  Call Extruder(272.17524)
  MoveL 6100 to (227.15, 164.34, 88.06) mm, rotated rx 180 ry 0 rz 180 deg; joints [-30.903, 18.099, 54.936, 64.012, 34.845, -59.291]
  MoveL 6101 to (227.15, 164.34, 88.06) mm, rotated rx 180 ry 0 rz 180 deg; joints [-30.903, 18.099, 54.936, 64.012, 34.845, -59.291]
  Call Extruder(272.32310)
  MoveL 6102 to (226.87, 164.39, 88.06) mm, rotated rx 180 ry 0 rz 180 deg; joints [-30.923, 18.056, 54.993, 64.047, 34.856, -59.326]
  MoveL 6103 to (226.87, 164.39, 88.06) mm, rotated rx 180 ry 0 rz 180 deg; joints [-30.923, 18.056, 54.993, 64.047, 34.856, -59.326]
  Call Extruder(272.48484)
  MoveL 6104 to (226.57, 164.44, 88.06) mm, rotated rx 180 ry 0 rz 180 deg; joints [-30.943, 18.008, 55.056, 64.085, 34.867, -59.365]
  MoveL 6105 to (226.57, 164.44, 88.06) mm, rotated rx 180 ry 0 rz 180 deg; joints [-30.943, 18.008, 55.056, 64.085, 34.867, -59.365]
  Call Extruder(272.64586)
  MoveL 6106 to (226.26, 164.49, 88.06) mm, rotated rx 180 ry 0 rz 180 deg; joints [-30.964, 17.96, 55.119, 64.122, 34.879, -59.404]
  MoveL 6107 to (226.26, 164.49, 88.06) mm, rotated rx 180 ry 0 rz 180 deg; joints [-30.964, 17.96, 55.119, 64.122, 34.879, -59.404]
  Call Extruder(272.80614)
  MoveL 6108 to (225.95, 164.53, 88.06) mm, rotated rx 180 ry 0 rz 180 deg; joints [-30.985, 17.912, 55.182, 64.16, 34.89, -59.442]
  MoveL 6109 to (225.95, 164.53, 88.06) mm, rotated rx 180 ry 0 rz 180 deg; joints [-30.985, 17.912, 55.182, 64.16, 34.89, -59.442]
  Call Extruder(272.96570)
  MoveL 6110 to (225.65, 164.58, 88.06) mm, rotated rx 180 ry 0 rz 180 deg; joints [-31.006, 17.864, 55.244, 64.198, 34.901, -59.481]
  MoveL 6111 to (225.65, 164.58, 88.06) mm, rotated rx 180 ry 0 rz 180 deg; joints [-31.006, 17.864, 55.244, 64.198, 34.901, -59.481]
  Call Extruder(273.12452)
  MoveL 6112 to (225.34, 164.63, 88.06) mm, rotated rx -180 ry 0 rz 180 deg; joints [-31.027, 17.817, 55.307, 64.235, 34.913, -59.519]
  MoveL 6113 to (225.34, 164.63, 88.06) mm, rotated rx -180 ry 0 rz 180 deg; joints [-31.027, 17.817, 55.307, 64.235, 34.913, -59.519]
  Call Extruder(273.30319)
  MoveL 6114 to (225, 164.68, 88.06) mm, rotated rx 180 ry 0 rz 180 deg; joints [-31.049, 17.762, 55.379, 64.278, 34.925, -59.563]
  MoveL 6115 to (225, 164.68, 88.06) mm, rotated rx 180 ry 0 rz 180 deg; joints [-31.049, 17.762, 55.379, 64.278, 34.925, -59.563]
  Call Extruder(273.50164)
  MoveL 6116 to (224.61, 164.72, 88.06) mm, rotated rx -180 ry 0 rz 180 deg; joints [-31.074, 17.7, 55.459, 64.324, 34.939, -59.611]
  MoveL 6117 to (224.61, 164.72, 88.06) mm, rotated rx -180 ry 0 rz 180 deg; joints [-31.074, 17.7, 55.459, 64.324, 34.939, -59.611]
  Call Extruder(273.69921)
  MoveL 6118 to (224.22, 164.77, 88.06) mm, rotated rx 180 ry 0 rz 180 deg; joints [-31.1, 17.638, 55.54, 64.371, 34.952, -59.659]
  MoveL 6119 to (224.22, 164.77, 88.06) mm, rotated rx 180 ry 0 rz 180 deg; joints [-31.1, 17.638, 55.54, 64.371, 34.952, -59.659]
  Call Extruder(273.89592)
  MoveL 6120 to (223.84, 164.82, 88.06) mm, rotated rx 180 ry 0 rz 180 deg; joints [-31.125, 17.576, 55.621, 64.417, 34.966, -59.706]
  MoveL 6121 to (223.84, 164.82, 88.06) mm, rotated rx 180 ry 0 rz 180 deg; joints [-31.125, 17.576, 55.621, 64.417, 34.966, -59.706]
  Call Extruder(274.09176)
  MoveL 6122 to (223.45, 164.86, 88.06) mm, rotated rx -180 ry 0 rz 180 deg; joints [-31.15, 17.514, 55.701, 64.463, 34.979, -59.754]
  MoveL 6123 to (223.45, 164.86, 88.06) mm, rotated rx -180 ry 0 rz 180 deg; joints [-31.15, 17.514, 55.701, 64.463, 34.979, -59.754]
  Call Extruder(274.38712)
  MoveL 6124 to (222.86, 164.91, 88.06) mm, rotated rx 180 ry 0 rz -180 deg; joints [-31.186, 17.419, 55.826, 64.533, 34.998, -59.826]
  MoveL 6125 to (222.86, 164.91, 88.06) mm, rotated rx 180 ry 0 rz -180 deg; joints [-31.186, 17.419, 55.826, 64.533, 34.998, -59.826]
  Call Extruder(274.68114)
  MoveL 6126 to (222.27, 164.96, 88.06) mm, rotated rx 180 ry 0 rz 180 deg; joints [-31.222, 17.323, 55.951, 64.601, 35.017, -59.897]
  MoveL 6127 to (222.27, 164.96, 88.06) mm, rotated rx 180 ry 0 rz 180 deg; joints [-31.222, 17.323, 55.951, 64.601, 35.017, -59.897]
  Call Extruder(274.97384)
  MoveL 6128 to (221.68, 165, 88.06) mm, rotated rx 180 ry 0 rz 180 deg; joints [-31.258, 17.227, 56.075, 64.67, 35.036, -59.968]
  MoveL 6129 to (221.68, 165, 88.06) mm, rotated rx 180 ry 0 rz 180 deg; joints [-31.258, 17.227, 56.075, 64.67, 35.036, -59.968]
  Call Extruder(275.54729)
  MoveL 6130 to (220.52, 165.05, 88.06) mm, rotated rx 180 ry 0 rz 180 deg; joints [-31.326, 17.035, 56.324, 64.802, 35.07, -60.106]
  MoveL 6131 to (220.52, 165.05, 88.06) mm, rotated rx 180 ry 0 rz 180 deg; joints [-31.326, 17.035, 56.324, 64.802, 35.07, -60.106]
  Call Extruder(276.26129)
  MoveL 6132 to (219.06, 165.09, 88.06) mm, rotated rx -180 ry 0 rz 180 deg; joints [-31.409, 16.794, 56.636, 64.966, 35.113, -60.277]
  Call Extruder(393.10803)
  MoveL 6133 to (-19.06, 165.09, 88.06) mm, rotated rx 180 ry 0 rz 180 deg; joints [-51.475, -12.583, 87.083, 77.988, 53.116, -70.481]
  Call Extruder(393.53664)
  MoveL 6134 to (-19.94, 165.07, 88.06) mm, rotated rx 180 ry 0 rz 180 deg; joints [-51.582, -12.664, 87.145, 78.02, 53.22, -70.486]
  MoveL 6135 to (-19.94, 165.07, 88.06) mm, rotated rx 180 ry 0 rz 180 deg; joints [-51.582, -12.664, 87.145, 78.02, 53.22, -70.486]
  Call Extruder(394.11009)
  MoveL 6136 to (-21.1, 165.03, 88.06) mm, rotated rx 180 ry 0 rz 180 deg; joints [-51.722, -12.772, 87.23, 78.061, 53.357, -70.492]
  MoveL 6137 to (-21.1, 165.03, 88.06) mm, rotated rx 180 ry 0 rz 180 deg; joints [-51.722, -12.772, 87.23, 78.061, 53.357, -70.492]
  Call Extruder(394.54439)
  MoveL 6138 to (-21.97, 164.98, 88.06) mm, rotated rx 180 ry 0 rz 180 deg; joints [-51.827, -12.855, 87.295, 78.091, 53.46, -70.495]
  MoveL 6139 to (-21.97, 164.98, 88.06) mm, rotated rx 180 ry 0 rz 180 deg; joints [-51.827, -12.855, 87.295, 78.091, 53.46, -70.495]
  Call Extruder(394.83842)
  MoveL 6140 to (-22.56, 164.93, 88.06) mm, rotated rx 180 ry 0 rz -180 deg; joints [-51.897, -12.913, 87.34, 78.111, 53.528, -70.497]
  MoveL 6141 to (-22.56, 164.93, 88.06) mm, rotated rx 180 ry 0 rz -180 deg; joints [-51.897, -12.913, 87.34, 78.111, 53.528, -70.497]
  Call Extruder(395.13378)
  MoveL 6142 to (-23.15, 164.89, 88.06) mm, rotated rx 180 ry 0 rz 180 deg; joints [-51.966, -12.97, 87.384, 78.131, 53.596, -70.499]
  MoveL 6143 to (-23.15, 164.89, 88.06) mm, rotated rx 180 ry 0 rz 180 deg; joints [-51.966, -12.97, 87.384, 78.131, 53.596, -70.499]
  Call Extruder(395.37999)
  MoveL 6144 to (-23.64, 164.84, 88.06) mm, rotated rx 180 ry 0 rz 180 deg; joints [-52.023, -13.018, 87.421, 78.146, 53.652, -70.499]
  MoveL 6145 to (-23.64, 164.84, 88.06) mm, rotated rx 180 ry 0 rz 180 deg; joints [-52.023, -13.018, 87.421, 78.146, 53.652, -70.499]
  Call Extruder(395.57670)
  MoveL 6146 to (-24.03, 164.79, 88.06) mm, rotated rx -180 ry 0 rz 180 deg; joints [-52.067, -13.058, 87.452, 78.158, 53.696, -70.499]
  MoveL 6147 to (-24.03, 164.79, 88.06) mm, rotated rx -180 ry 0 rz 180 deg; joints [-52.067, -13.058, 87.452, 78.158, 53.696, -70.499]
  Call Extruder(395.77427)
  MoveL 6148 to (-24.42, 164.75, 88.06) mm, rotated rx 180 ry 0 rz 180 deg; joints [-52.112, -13.097, 87.482, 78.17, 53.739, -70.5]
  MoveL 6149 to (-24.42, 164.75, 88.06) mm, rotated rx 180 ry 0 rz 180 deg; joints [-52.112, -13.097, 87.482, 78.17, 53.739, -70.5]
  Call Extruder(395.97271)
  MoveL 6150 to (-24.8, 164.7, 88.06) mm, rotated rx 180 ry 0 rz 180 deg; joints [-52.156, -13.136, 87.513, 78.182, 53.783, -70.5]
  MoveL 6151 to (-24.8, 164.7, 88.06) mm, rotated rx 180 ry 0 rz 180 deg; joints [-52.156, -13.136, 87.513, 78.182, 53.783, -70.5]
  Call Extruder(396.17202)
  MoveL 6152 to (-25.19, 164.66, 88.06) mm, rotated rx 180 ry 0 rz 180 deg; joints [-52.2, -13.176, 87.543, 78.194, 53.827, -70.5]
  MoveL 6153 to (-25.19, 164.66, 88.06) mm, rotated rx 180 ry 0 rz 180 deg; joints [-52.2, -13.176, 87.543, 78.194, 53.827, -70.5]
  Call Extruder(396.33085)
  MoveL 6154 to (-25.5, 164.61, 88.06) mm, rotated rx 180 ry 0 rz 180 deg; joints [-52.235, -13.208, 87.568, 78.203, 53.86, -70.499]
  MoveL 6155 to (-25.5, 164.61, 88.06) mm, rotated rx 180 ry 0 rz 180 deg; joints [-52.235, -13.208, 87.568, 78.203, 53.86, -70.499]
  Call Extruder(396.49041)
  MoveL 6156 to (-25.8, 164.56, 88.06) mm, rotated rx 180 ry 0 rz 180 deg; joints [-52.269, -13.24, 87.593, 78.212, 53.894, -70.498]
  MoveL 6157 to (-25.8, 164.56, 88.06) mm, rotated rx 180 ry 0 rz 180 deg; joints [-52.269, -13.24, 87.593, 78.212, 53.894, -70.498]
  Call Extruder(396.65070)
  MoveL 6158 to (-26.11, 164.51, 88.06) mm, rotated rx 180 ry 0 rz -180 deg; joints [-52.303, -13.272, 87.618, 78.221, 53.927, -70.498]
  MoveL 6159 to (-26.11, 164.51, 88.06) mm, rotated rx 180 ry 0 rz -180 deg; joints [-52.303, -13.272, 87.618, 78.221, 53.927, -70.498]
  Call Extruder(396.81172)
  MoveL 6160 to (-26.41, 164.46, 88.06) mm, rotated rx 180 ry 0 rz -180 deg; joints [-52.337, -13.305, 87.643, 78.229, 53.961, -70.497]
  MoveL 6161 to (-26.41, 164.46, 88.06) mm, rotated rx 180 ry 0 rz -180 deg; joints [-52.337, -13.305, 87.643, 78.229, 53.961, -70.497]
  Call Extruder(396.97346)
  MoveL 6162 to (-26.72, 164.41, 88.06) mm, rotated rx -180 ry 0 rz 180 deg; joints [-52.371, -13.337, 87.668, 78.238, 53.995, -70.496]
  MoveL 6163 to (-26.72, 164.41, 88.06) mm, rotated rx -180 ry 0 rz 180 deg; joints [-52.371, -13.337, 87.668, 78.238, 53.995, -70.496]
  Call Extruder(397.13593)
  MoveL 6164 to (-27.02, 164.37, 88.06) mm, rotated rx 180 ry 0 rz -180 deg; joints [-52.405, -13.369, 87.692, 78.247, 54.028, -70.496]
  MoveL 6165 to (-27.02, 164.37, 88.06) mm, rotated rx 180 ry 0 rz -180 deg; joints [-52.405, -13.369, 87.692, 78.247, 54.028, -70.496]
  Call Extruder(397.26986)
  MoveL 6166 to (-27.27, 164.32, 88.06) mm, rotated rx 180 ry 0 rz 180 deg; joints [-52.432, -13.397, 87.713, 78.254, 54.055, -70.495]
  MoveL 6167 to (-27.27, 164.32, 88.06) mm, rotated rx 180 ry 0 rz 180 deg; joints [-52.432, -13.397, 87.713, 78.254, 54.055, -70.495]
  Call Extruder(397.40439)
  MoveL 6168 to (-27.52, 164.27, 88.06) mm, rotated rx 180 ry 0 rz 180 deg; joints [-52.459, -13.424, 87.734, 78.26, 54.082, -70.493]
  MoveL 6169 to (-27.52, 164.27, 88.06) mm, rotated rx 180 ry 0 rz 180 deg; joints [-52.459, -13.424, 87.734, 78.26, 54.082, -70.493]
  Call Extruder(397.53954)
  MoveL 6170 to (-27.77, 164.22, 88.06) mm, rotated rx 180 ry 0 rz 180 deg; joints [-52.486, -13.451, 87.755, 78.267, 54.109, -70.492]
  MoveL 6171 to (-27.77, 164.22, 88.06) mm, rotated rx 180 ry 0 rz 180 deg; joints [-52.486, -13.451, 87.755, 78.267, 54.109, -70.492]
  Call Extruder(397.67530)
  MoveL 6172 to (-28.02, 164.17, 88.06) mm, rotated rx 180 ry 0 rz -180 deg; joints [-52.513, -13.479, 87.776, 78.274, 54.135, -70.491]
  MoveL 6173 to (-28.02, 164.17, 88.06) mm, rotated rx 180 ry 0 rz -180 deg; joints [-52.513, -13.479, 87.776, 78.274, 54.135, -70.491]
  Call Extruder(397.81166)
  MoveL 6174 to (-28.27, 164.12, 88.06) mm, rotated rx 180 ry 0 rz 180 deg; joints [-52.54, -13.506, 87.797, 78.28, 54.162, -70.49]
  MoveL 6175 to (-28.27, 164.12, 88.06) mm, rotated rx 180 ry 0 rz 180 deg; joints [-52.54, -13.506, 87.797, 78.28, 54.162, -70.49]
  Call Extruder(397.89653)
  MoveL 6176 to (-28.43, 164.09, 88.06) mm, rotated rx -180 ry 0 rz -180 deg; joints [-52.556, -13.523, 87.81, 78.284, 54.179, -70.489]
  Set speed (130.0 mm/s)
  MoveL 6177 to (-31.76, 163.31, 88.06) mm, rotated rx 180 ry 0 rz 180 deg; joints [-52.91, -13.899, 88.098, 78.367, 54.529, -70.466]
  MoveL 6178 to (-31.76, 163.31, 97.46) mm, rotated rx 180 ry 0 rz 180 deg; joints [-52.91, -14.605, 90.097, 79.276, 54.279, -72.028]
  Call Extruder(395.89653)
  Set speed (40.0 mm/s)
  MoveL 6179 to (-31.76, 163.31, 97.46) mm, rotated rx 180 ry 0 rz 180 deg; joints [-52.91, -14.605, 90.097, 79.276, 54.279, -72.028]
  Call Extruder(0.00000)
  Set speed (130.0 mm/s)
  MoveL 6180 to (-31.64, 163.21, 97.46) mm, rotated rx 180 ry 0 rz 180 deg; joints [-52.884, -14.606, 90.098, 79.266, 54.254, -72.022]
  Call Extruder(2.00000)
  Set speed (40.0 mm/s)
  MoveL 6181 to (-31.64, 163.21, 97.46) mm, rotated rx 180 ry 0 rz 180 deg; joints [-52.884, -14.606, 90.098, 79.266, 54.254, -72.022]
  Set speed (30.0 mm/s)
  MoveL 6182 to (-31.64, 163.21, 97.46) mm, rotated rx 180 ry 0 rz 180 deg; joints [-52.884, -14.606, 90.098, 79.266, 54.254, -72.022]
  Call Extruder(2.18198)
  MoveL 6183 to (-31.93, 163.09, 97.46) mm, rotated rx -180 ry 0 rz 180 deg; joints [-52.91, -14.645, 90.127, 79.269, 54.281, -72.016]
  MoveL 6184 to (-31.93, 163.09, 97.46) mm, rotated rx -180 ry 0 rz 180 deg; joints [-52.91, -14.645, 90.127, 79.269, 54.281, -72.016]
  Call Extruder(2.36471)
  MoveL 6185 to (-32.22, 162.97, 97.46) mm, rotated rx 180 ry 0 rz 180 deg; joints [-52.936, -14.684, 90.157, 79.272, 54.307, -72.01]
  MoveL 6186 to (-32.22, 162.97, 97.46) mm, rotated rx 180 ry 0 rz 180 deg; joints [-52.936, -14.684, 90.157, 79.272, 54.307, -72.01]
  Call Extruder(2.53513)
  MoveL 6187 to (-32.49, 162.85, 97.46) mm, rotated rx 180 ry 0 rz 180 deg; joints [-52.96, -14.72, 90.184, 79.275, 54.332, -72.004]
  MoveL 6188 to (-32.49, 162.85, 97.46) mm, rotated rx 180 ry 0 rz 180 deg; joints [-52.96, -14.72, 90.184, 79.275, 54.332, -72.004]
  Call Extruder(2.69310)
  MoveL 6189 to (-32.74, 162.74, 97.46) mm, rotated rx 180 ry 0 rz 180 deg; joints [-52.982, -14.754, 90.209, 79.277, 54.354, -71.999]
  MoveL 6190 to (-32.74, 162.74, 97.46) mm, rotated rx 180 ry 0 rz 180 deg; joints [-52.982, -14.754, 90.209, 79.277, 54.354, -71.999]
  Call Extruder(2.85168)
  MoveL 6191 to (-32.99, 162.64, 97.46) mm, rotated rx 180 ry 0 rz 180 deg; joints [-53.004, -14.788, 90.234, 79.279, 54.377, -71.993]
  MoveL 6192 to (-32.99, 162.64, 97.46) mm, rotated rx 180 ry 0 rz 180 deg; joints [-53.004, -14.788, 90.234, 79.279, 54.377, -71.993]
  Call Extruder(3.05785)
  MoveL 6193 to (-33.29, 162.46, 97.46) mm, rotated rx 180 ry 0 rz 180 deg; joints [-53.026, -14.834, 90.269, 79.28, 54.4, -71.984]
  MoveL 6194 to (-33.29, 162.46, 97.46) mm, rotated rx 180 ry 0 rz 180 deg; joints [-53.026, -14.834, 90.269, 79.28, 54.4, -71.984]
  Call Extruder(3.26479)
  MoveL 6195 to (-33.6, 162.29, 97.46) mm, rotated rx 180 ry 0 rz 180 deg; joints [-53.049, -14.88, 90.303, 79.28, 54.424, -71.975]
  MoveL 6196 to (-33.6, 162.29, 97.46) mm, rotated rx 180 ry 0 rz 180 deg; joints [-53.049, -14.88, 90.303, 79.28, 54.424, -71.975]
  Call Extruder(3.47251)
  MoveL 6197 to (-33.9, 162.11, 97.46) mm, rotated rx 180 ry 0 rz 180 deg; joints [-53.071, -14.926, 90.338, 79.28, 54.447, -71.966]
  MoveL 6198 to (-33.9, 162.11, 97.46) mm, rotated rx 180 ry 0 rz 180 deg; joints [-53.071, -14.926, 90.338, 79.28, 54.447, -71.966]
  Call Extruder(3.68101)
  MoveL 6199 to (-34.21, 161.93, 97.46) mm, rotated rx -180 ry 0 rz -180 deg; joints [-53.094, -14.972, 90.372, 79.281, 54.471, -71.957]
  MoveL 6200 to (-34.21, 161.93, 97.46) mm, rotated rx -180 ry 0 rz -180 deg; joints [-53.094, -14.972, 90.372, 79.281, 54.471, -71.957]
  Call Extruder(3.86055)
  MoveL 6201 to (-34.45, 161.76, 97.46) mm, rotated rx 180 ry 0 rz -180 deg; joints [-53.109, -15.013, 90.403, 79.279, 54.487, -71.947]
  MoveL 6202 to (-34.45, 161.76, 97.46) mm, rotated rx 180 ry 0 rz -180 deg; joints [-53.109, -15.013, 90.403, 79.279, 54.487, -71.947]
  Call Extruder(4.19399)
  MoveL 6203 to (-34.9, 161.43, 97.46) mm, rotated rx 180 ry 0 rz 180 deg; joints [-53.135, -15.09, 90.459, 79.275, 54.516, -71.93]
  MoveL 6204 to (-34.9, 161.43, 97.46) mm, rotated rx 180 ry 0 rz 180 deg; joints [-53.135, -15.09, 90.459, 79.275, 54.516, -71.93]
  Call Extruder(4.52861)
  MoveL 6205 to (-35.35, 161.1, 97.46) mm, rotated rx 180 ry 0 rz 180 deg; joints [-53.163, -15.166, 90.516, 79.272, 54.546, -71.912]
  Call Extruder(5.35652)
  MoveL 6206 to (-36.39, 160.19, 97.46) mm, rotated rx 180 ry 0 rz 180 deg; joints [-53.209, -15.359, 90.659, 79.255, 54.599, -71.862]
  Call Extruder(6.18445)
  MoveL 6207 to (-37.3, 159.15, 97.46) mm, rotated rx 180 ry 0 rz 180 deg; joints [-53.227, -15.555, 90.803, 79.225, 54.626, -71.803]
  Call Extruder(6.35176)
  MoveL 6208 to (-37.47, 158.93, 97.46) mm, rotated rx 180 ry 0 rz 180 deg; joints [-53.227, -15.595, 90.832, 79.218, 54.628, -71.79]
  MoveL 6209 to (-37.47, 158.93, 97.46) mm, rotated rx 180 ry 0 rz 180 deg; joints [-53.227, -15.595, 90.832, 79.218, 54.628, -71.79]
  Call Extruder(6.68519)
  MoveL 6210 to (-37.79, 158.48, 97.46) mm, rotated rx -180 ry 0 rz 180 deg; joints [-53.226, -15.674, 90.89, 79.203, 54.63, -71.765]
  MoveL 6211 to (-37.79, 158.48, 97.46) mm, rotated rx -180 ry 0 rz 180 deg; joints [-53.226, -15.674, 90.89, 79.203, 54.63, -71.765]
  Call Extruder(7.01743)
  MoveL 6212 to (-38.12, 158.03, 97.46) mm, rotated rx 180 ry 0 rz 180 deg; joints [-53.224, -15.754, 90.949, 79.187, 54.633, -71.739]
  MoveL 6213 to (-38.12, 158.03, 97.46) mm, rotated rx 180 ry 0 rz 180 deg; joints [-53.224, -15.754, 90.949, 79.187, 54.633, -71.739]
  Call Extruder(7.13511)
  MoveL 6214 to (-38.22, 157.85, 97.46) mm, rotated rx 180 ry 0 rz 180 deg; joints [-53.221, -15.782, 90.969, 79.181, 54.631, -71.729]
  MoveL 6215 to (-38.22, 157.85, 97.46) mm, rotated rx 180 ry 0 rz 180 deg; joints [-53.221, -15.782, 90.969, 79.181, 54.631, -71.729]
  Call Extruder(7.34283)
  MoveL 6216 to (-38.4, 157.55, 97.46) mm, rotated rx -180 ry 0 rz 180 deg; joints [-53.214, -15.831, 91.005, 79.169, 54.627, -71.711]
  MoveL 6217 to (-38.4, 157.55, 97.46) mm, rotated rx -180 ry 0 rz 180 deg; joints [-53.214, -15.831, 91.005, 79.169, 54.627, -71.711]
  Call Extruder(7.54978)
  MoveL 6218 to (-38.57, 157.25, 97.46) mm, rotated rx 180 ry 0 rz 180 deg; joints [-53.207, -15.881, 91.042, 79.157, 54.623, -71.693]
  MoveL 6219 to (-38.57, 157.25, 97.46) mm, rotated rx 180 ry 0 rz 180 deg; joints [-53.207, -15.881, 91.042, 79.157, 54.623, -71.693]
  Call Extruder(7.75595)
  MoveL 6220 to (-38.75, 156.94, 97.46) mm, rotated rx 180 ry 0 rz 180 deg; joints [-53.2, -15.93, 91.078, 79.144, 54.619, -71.676]
  MoveL 6221 to (-38.75, 156.94, 97.46) mm, rotated rx 180 ry 0 rz 180 deg; joints [-53.2, -15.93, 91.078, 79.144, 54.619, -71.676]
  Call Extruder(7.93762)
  MoveL 6222 to (-38.89, 156.67, 97.46) mm, rotated rx 180 ry 0 rz 180 deg; joints [-53.191, -15.974, 91.109, 79.133, 54.613, -71.659]
  MoveL 6223 to (-38.89, 156.67, 97.46) mm, rotated rx 180 ry 0 rz 180 deg; joints [-53.191, -15.974, 91.109, 79.133, 54.613, -71.659]
  Call Extruder(8.09561)
  MoveL 6224 to (-39, 156.42, 97.46) mm, rotated rx 180 ry 0 rz 180 deg; joints [-53.18, -16.011, 91.137, 79.122, 54.605, -71.645]
  MoveL 6225 to (-39, 156.42, 97.46) mm, rotated rx 180 ry 0 rz 180 deg; joints [-53.18, -16.011, 91.137, 79.122, 54.605, -71.645]
  Call Extruder(8.25299)
  MoveL 6226 to (-39.1, 156.17, 97.46) mm, rotated rx 180 ry 0 rz 180 deg; joints [-53.17, -16.049, 91.164, 79.11, 54.596, -71.63]
  MoveL 6227 to (-39.1, 156.17, 97.46) mm, rotated rx 180 ry 0 rz 180 deg; joints [-53.17, -16.049, 91.164, 79.11, 54.596, -71.63]
  Call Extruder(8.43571)
  MoveL 6228 to (-39.23, 155.88, 97.46) mm, rotated rx 180 ry 0 rz 180 deg; joints [-53.156, -16.092, 91.195, 79.097, 54.586, -71.613]
  MoveL 6229 to (-39.23, 155.88, 97.46) mm, rotated rx 180 ry 0 rz 180 deg; joints [-53.156, -16.092, 91.195, 79.097, 54.586, -71.613]
  Call Extruder(8.61768)
  MoveL 6230 to (-39.35, 155.58, 97.46) mm, rotated rx 180 ry 0 rz 180 deg; joints [-53.143, -16.136, 91.227, 79.083, 54.576, -71.595]
  MoveL 6231 to (-39.35, 155.58, 97.46) mm, rotated rx 180 ry 0 rz 180 deg; joints [-53.143, -16.136, 91.227, 79.083, 54.576, -71.595]
  Call Extruder(8.76501)
  MoveL 6232 to (-39.44, 155.34, 97.46) mm, rotated rx 180 ry 0 rz 180 deg; joints [-53.131, -16.171, 91.252, 79.072, 54.566, -71.581]
  MoveL 6233 to (-39.44, 155.34, 97.46) mm, rotated rx 180 ry 0 rz 180 deg; joints [-53.131, -16.171, 91.252, 79.072, 54.566, -71.581]
  Call Extruder(8.87824)
  MoveL 6234 to (-39.5, 155.15, 97.46) mm, rotated rx 180 ry 0 rz 180 deg; joints [-53.121, -16.198, 91.272, 79.063, 54.558, -71.57]
  MoveL 6235 to (-39.5, 155.15, 97.46) mm, rotated rx 180 ry 0 rz 180 deg; joints [-53.121, -16.198, 91.272, 79.063, 54.558, -71.57]
  Call Extruder(8.99103)
  MoveL 6236 to (-39.56, 154.97, 97.46) mm, rotated rx 180 ry 0 rz 180 deg; joints [-53.11, -16.224, 91.291, 79.053, 54.549, -71.558]
  MoveL 6237 to (-39.56, 154.97, 97.46) mm, rotated rx 180 ry 0 rz 180 deg; joints [-53.11, -16.224, 91.291, 79.053, 54.549, -71.558]
  Call Extruder(9.10338)
  MoveL 6238 to (-39.62, 154.78, 97.46) mm, rotated rx -180 ry 0 rz -180 deg; joints [-53.099, -16.251, 91.31, 79.044, 54.54, -71.547]
  MoveL 6239 to (-39.62, 154.78, 97.46) mm, rotated rx -180 ry 0 rz -180 deg; joints [-53.099, -16.251, 91.31, 79.044, 54.54, -71.547]
  Call Extruder(9.21528)
  MoveL 6240 to (-39.68, 154.59, 97.46) mm, rotated rx 180 ry 0 rz 180 deg; joints [-53.088, -16.277, 91.329, 79.035, 54.531, -71.536]
  MoveL 6241 to (-39.68, 154.59, 97.46) mm, rotated rx 180 ry 0 rz 180 deg; joints [-53.088, -16.277, 91.329, 79.035, 54.531, -71.536]
  Call Extruder(9.33668)
  MoveL 6242 to (-39.75, 154.38, 97.46) mm, rotated rx -180 ry 0 rz 180 deg; joints [-53.076, -16.306, 91.35, 79.024, 54.521, -71.523]
  MoveL 6243 to (-39.75, 154.38, 97.46) mm, rotated rx -180 ry 0 rz 180 deg; joints [-53.076, -16.306, 91.35, 79.024, 54.521, -71.523]
  Call Extruder(9.46747)
  MoveL 6244 to (-39.81, 154.16, 97.46) mm, rotated rx 180 ry 0 rz 180 deg; joints [-53.063, -16.337, 91.373, 79.013, 54.51, -71.51]
  MoveL 6245 to (-39.81, 154.16, 97.46) mm, rotated rx 180 ry 0 rz 180 deg; joints [-53.063, -16.337, 91.373, 79.013, 54.51, -71.51]
  Call Extruder(9.59770)
  MoveL 6246 to (-39.88, 153.94, 97.46) mm, rotated rx 180 ry 0 rz 180 deg; joints [-53.049, -16.368, 91.395, 79.002, 54.499, -71.496]
  MoveL 6247 to (-39.88, 153.94, 97.46) mm, rotated rx 180 ry 0 rz 180 deg; joints [-53.049, -16.368, 91.395, 79.002, 54.499, -71.496]
  Call Extruder(9.72737)
  MoveL 6248 to (-39.95, 153.71, 97.46) mm, rotated rx -180 ry 0 rz -180 deg; joints [-53.036, -16.4, 91.417, 78.99, 54.488, -71.482]
  MoveL 6249 to (-39.95, 153.71, 97.46) mm, rotated rx -180 ry 0 rz -180 deg; joints [-53.036, -16.4, 91.417, 78.99, 54.488, -71.482]
  Call Extruder(9.85647)
  MoveL 6250 to (-40.02, 153.49, 97.46) mm, rotated rx -180 ry 0 rz 180 deg; joints [-53.022, -16.431, 91.44, 78.979, 54.476, -71.469]
  MoveL 6251 to (-40.02, 153.49, 97.46) mm, rotated rx -180 ry 0 rz 180 deg; joints [-53.022, -16.431, 91.44, 78.979, 54.476, -71.469]
  Call Extruder(9.97155)
  MoveL 6252 to (-40.06, 153.28, 97.46) mm, rotated rx 180 ry 0 rz 180 deg; joints [-53.007, -16.458, 91.459, 78.968, 54.464, -71.456]
  MoveL 6253 to (-40.06, 153.28, 97.46) mm, rotated rx 180 ry 0 rz 180 deg; joints [-53.007, -16.458, 91.459, 78.968, 54.464, -71.456]
  Call Extruder(10.08619)
  MoveL 6254 to (-40.11, 153.08, 97.46) mm, rotated rx 180 ry 0 rz 180 deg; joints [-52.993, -16.485, 91.479, 78.957, 54.452, -71.444]
  MoveL 6255 to (-40.11, 153.08, 97.46) mm, rotated rx 180 ry 0 rz 180 deg; joints [-52.993, -16.485, 91.479, 78.957, 54.452, -71.444]
  Call Extruder(10.20037)
  MoveL 6256 to (-40.15, 152.88, 97.46) mm, rotated rx 180 ry 0 rz 180 deg; joints [-52.978, -16.512, 91.498, 78.946, 54.439, -71.431]
  MoveL 6257 to (-40.15, 152.88, 97.46) mm, rotated rx 180 ry 0 rz 180 deg; joints [-52.978, -16.512, 91.498, 78.946, 54.439, -71.431]
  Call Extruder(10.31410)
  MoveL 6258 to (-40.2, 152.67, 97.46) mm, rotated rx -180 ry 0 rz 180 deg; joints [-52.963, -16.539, 91.517, 78.935, 54.426, -71.419]
  MoveL 6259 to (-40.2, 152.67, 97.46) mm, rotated rx -180 ry 0 rz 180 deg; joints [-52.963, -16.539, 91.517, 78.935, 54.426, -71.419]
  Call Extruder(10.43952)
  MoveL 6260 to (-40.24, 152.45, 97.46) mm, rotated rx -180 ry 0 rz 180 deg; joints [-52.946, -16.568, 91.539, 78.922, 54.412, -71.405]
  MoveL 6261 to (-40.24, 152.45, 97.46) mm, rotated rx -180 ry 0 rz 180 deg; joints [-52.946, -16.568, 91.539, 78.922, 54.412, -71.405]
  Call Extruder(10.57650)
  MoveL 6262 to (-40.29, 152.2, 97.46) mm, rotated rx -180 ry 0 rz 180 deg; joints [-52.928, -16.601, 91.562, 78.908, 54.396, -71.39]
  MoveL 6263 to (-40.29, 152.2, 97.46) mm, rotated rx -180 ry 0 rz 180 deg; joints [-52.928, -16.601, 91.562, 78.908, 54.396, -71.39]
  Call Extruder(10.71287)
  MoveL 6264 to (-40.34, 151.95, 97.46) mm, rotated rx -180 ry 0 rz -180 deg; joints [-52.909, -16.633, 91.585, 78.894, 54.38, -71.374]
  MoveL 6265 to (-40.34, 151.95, 97.46) mm, rotated rx -180 ry 0 rz -180 deg; joints [-52.909, -16.633, 91.585, 78.894, 54.38, -71.374]
  Call Extruder(10.84862)
  MoveL 6266 to (-40.39, 151.7, 97.46) mm, rotated rx 180 ry 0 rz 180 deg; joints [-52.89, -16.665, 91.608, 78.881, 54.364, -71.359]
  MoveL 6267 to (-40.39, 151.7, 97.46) mm, rotated rx 180 ry 0 rz 180 deg; joints [-52.89, -16.665, 91.608, 78.881, 54.364, -71.359]
  Call Extruder(10.98377)
  MoveL 6268 to (-40.44, 151.45, 97.46) mm, rotated rx -180 ry 0 rz -180 deg; joints [-52.871, -16.698, 91.631, 78.867, 54.348, -71.343]
  MoveL 6269 to (-40.44, 151.45, 97.46) mm, rotated rx -180 ry 0 rz -180 deg; joints [-52.871, -16.698, 91.631, 78.867, 54.348, -71.343]
  Call Extruder(11.11830)
  MoveL 6270 to (-40.49, 151.2, 97.46) mm, rotated rx 180 ry 0 rz 180 deg; joints [-52.853, -16.73, 91.654, 78.853, 54.332, -71.328]
  MoveL 6271 to (-40.49, 151.2, 97.46) mm, rotated rx 180 ry 0 rz 180 deg; joints [-52.853, -16.73, 91.654, 78.853, 54.332, -71.328]
  Call Extruder(11.25223)
  MoveL 6272 to (-40.54, 150.95, 97.46) mm, rotated rx 180 ry 0 rz 180 deg; joints [-52.834, -16.762, 91.678, 78.839, 54.316, -71.312]
  MoveL 6273 to (-40.54, 150.95, 97.46) mm, rotated rx 180 ry 0 rz 180 deg; joints [-52.834, -16.762, 91.678, 78.839, 54.316, -71.312]
  Call Extruder(11.40008)
  MoveL 6274 to (-40.59, 150.67, 97.46) mm, rotated rx 180 ry 0 rz 180 deg; joints [-52.812, -16.798, 91.703, 78.823, 54.297, -71.295]
  MoveL 6275 to (-40.59, 150.67, 97.46) mm, rotated rx 180 ry 0 rz 180 deg; joints [-52.812, -16.798, 91.703, 78.823, 54.297, -71.295]
  Call Extruder(11.56181)
  MoveL 6276 to (-40.64, 150.37, 97.46) mm, rotated rx 180 ry 0 rz 180 deg; joints [-52.787, -16.837, 91.73, 78.805, 54.276, -71.276]
  MoveL 6277 to (-40.64, 150.37, 97.46) mm, rotated rx 180 ry 0 rz 180 deg; joints [-52.787, -16.837, 91.73, 78.805, 54.276, -71.276]
  Call Extruder(11.72281)
  MoveL 6278 to (-40.69, 150.06, 97.46) mm, rotated rx 180 ry 0 rz -180 deg; joints [-52.762, -16.875, 91.758, 78.788, 54.254, -71.257]
  MoveL 6279 to (-40.69, 150.06, 97.46) mm, rotated rx 180 ry 0 rz -180 deg; joints [-52.762, -16.875, 91.758, 78.788, 54.254, -71.257]
  Call Extruder(11.88308)
  MoveL 6280 to (-40.73, 149.76, 97.46) mm, rotated rx -180 ry 0 rz 180 deg; joints [-52.737, -16.914, 91.785, 78.77, 54.233, -71.237]
  MoveL 6281 to (-40.73, 149.76, 97.46) mm, rotated rx -180 ry 0 rz 180 deg; joints [-52.737, -16.914, 91.785, 78.77, 54.233, -71.237]
  Call Extruder(12.04262)
  MoveL 6282 to (-40.78, 149.45, 97.46) mm, rotated rx 180 ry 0 rz 180 deg; joints [-52.712, -16.952, 91.813, 78.752, 54.212, -71.218]
  MoveL 6283 to (-40.78, 149.45, 97.46) mm, rotated rx 180 ry 0 rz 180 deg; joints [-52.712, -16.952, 91.813, 78.752, 54.212, -71.218]
  Call Extruder(12.20144)
  MoveL 6284 to (-40.83, 149.14, 97.46) mm, rotated rx 180 ry 0 rz 180 deg; joints [-52.687, -16.991, 91.84, 78.734, 54.19, -71.199]
  MoveL 6285 to (-40.83, 149.14, 97.46) mm, rotated rx 180 ry 0 rz 180 deg; joints [-52.687, -16.991, 91.84, 78.734, 54.19, -71.199]
  Call Extruder(12.38010)
  MoveL 6286 to (-40.88, 148.8, 97.46) mm, rotated rx 180 ry 0 rz 180 deg; joints [-52.658, -17.034, 91.871, 78.714, 54.165, -71.177]
  MoveL 6287 to (-40.88, 148.8, 97.46) mm, rotated rx 180 ry 0 rz 180 deg; joints [-52.658, -17.034, 91.871, 78.714, 54.165, -71.177]
  Call Extruder(12.57854)
  MoveL 6288 to (-40.93, 148.41, 97.46) mm, rotated rx -180 ry 0 rz 180 deg; joints [-52.624, -17.082, 91.904, 78.69, 54.135, -71.152]
  MoveL 6289 to (-40.93, 148.41, 97.46) mm, rotated rx -180 ry 0 rz 180 deg; joints [-52.624, -17.082, 91.904, 78.69, 54.135, -71.152]
  Call Extruder(12.77611)
  MoveL 6290 to (-40.97, 148.02, 97.46) mm, rotated rx -180 ry 0 rz -180 deg; joints [-52.59, -17.129, 91.938, 78.667, 54.106, -71.127]
  MoveL 6291 to (-40.97, 148.02, 97.46) mm, rotated rx -180 ry 0 rz -180 deg; joints [-52.59, -17.129, 91.938, 78.667, 54.106, -71.127]
  Call Extruder(12.97282)
  MoveL 6292 to (-41.02, 147.63, 97.46) mm, rotated rx 180 ry 0 rz 180 deg; joints [-52.556, -17.176, 91.971, 78.644, 54.076, -71.103]
  MoveL 6293 to (-41.02, 147.63, 97.46) mm, rotated rx 180 ry 0 rz 180 deg; joints [-52.556, -17.176, 91.971, 78.644, 54.076, -71.103]
  Call Extruder(13.16866)
  MoveL 6294 to (-41.06, 147.25, 97.46) mm, rotated rx 180 ry 0 rz -180 deg; joints [-52.521, -17.224, 92.005, 78.62, 54.047, -71.078]
  MoveL 6295 to (-41.06, 147.25, 97.46) mm, rotated rx 180 ry 0 rz -180 deg; joints [-52.521, -17.224, 92.005, 78.62, 54.047, -71.078]
  Call Extruder(13.46406)
  MoveL 6296 to (-41.11, 146.66, 97.46) mm, rotated rx -180 ry 0 rz 180 deg; joints [-52.466, -17.294, 92.054, 78.583, 53.999, -71.04]
  MoveL 6297 to (-41.11, 146.66, 97.46) mm, rotated rx -180 ry 0 rz 180 deg; joints [-52.466, -17.294, 92.054, 78.583, 53.999, -71.04]
  Call Extruder(13.75812)
  MoveL 6298 to (-41.16, 146.07, 97.46) mm, rotated rx 180 ry 0 rz 180 deg; joints [-52.411, -17.364, 92.104, 78.546, 53.95, -71.001]
  MoveL 6299 to (-41.16, 146.07, 97.46) mm, rotated rx 180 ry 0 rz 180 deg; joints [-52.411, -17.364, 92.104, 78.546, 53.95, -71.001]
  Call Extruder(14.05086)
  MoveL 6300 to (-41.2, 145.48, 97.46) mm, rotated rx -180 ry 0 rz 180 deg; joints [-52.355, -17.434, 92.153, 78.509, 53.902, -70.963]
  MoveL 6301 to (-41.2, 145.48, 97.46) mm, rotated rx -180 ry 0 rz 180 deg; joints [-52.355, -17.434, 92.153, 78.509, 53.902, -70.963]
  Call Extruder(14.62431)
  MoveL 6302 to (-41.25, 144.32, 97.46) mm, rotated rx 180 ry 0 rz 180 deg; joints [-52.239, -17.568, 92.246, 78.433, 53.8, -70.887]
  MoveL 6303 to (-41.25, 144.32, 97.46) mm, rotated rx 180 ry 0 rz 180 deg; joints [-52.239, -17.568, 92.246, 78.433, 53.8, -70.887]
  Call Extruder(15.33827)
  MoveL 6304 to (-41.29, 142.86, 97.46) mm, rotated rx 180 ry 0 rz 180 deg; joints [-52.09, -17.733, 92.362, 78.336, 53.669, -70.79]
  Call Extruder(57.40309)
  MoveL 6305 to (-41.29, 57.14, 97.46) mm, rotated rx -180 ry 0 rz 180 deg; joints [-40.759, -26.338, 97.705, 69.661, 44.13, -62.686]
  Call Extruder(57.83164)
  MoveL 6306 to (-41.27, 56.26, 97.46) mm, rotated rx -180 ry 0 rz -180 deg; joints [-40.614, -26.413, 97.746, 69.532, 44.014, -62.571]
  MoveL 6307 to (-41.27, 56.26, 97.46) mm, rotated rx -180 ry 0 rz -180 deg; joints [-40.614, -26.413, 97.746, 69.532, 44.014, -62.571]
  Call Extruder(58.11773)
  MoveL 6308 to (-41.25, 55.68, 97.46) mm, rotated rx 180 ry 0 rz 180 deg; joints [-40.517, -26.462, 97.773, 69.446, 43.935, -62.494]
  MoveL 6309 to (-41.25, 55.68, 97.46) mm, rotated rx 180 ry 0 rz 180 deg; joints [-40.517, -26.462, 97.773, 69.446, 43.935, -62.494]
  Call Extruder(58.69247)
  MoveL 6310 to (-41.2, 54.52, 97.46) mm, rotated rx 180 ry 0 rz 180 deg; joints [-40.32, -26.559, 97.825, 69.271, 43.776, -62.34]
  MoveL 6311 to (-41.2, 54.52, 97.46) mm, rotated rx 180 ry 0 rz 180 deg; joints [-40.32, -26.559, 97.825, 69.271, 43.776, -62.34]
  Call Extruder(58.98586)
  MoveL 6312 to (-41.15, 53.93, 97.46) mm, rotated rx 180 ry 0 rz 180 deg; joints [-40.217, -26.605, 97.85, 69.181, 43.693, -62.261]
  MoveL 6313 to (-41.15, 53.93, 97.46) mm, rotated rx 180 ry 0 rz 180 deg; joints [-40.217, -26.605, 97.85, 69.181, 43.693, -62.261]
  Call Extruder(59.28059)
  MoveL 6314 to (-41.11, 53.34, 97.46) mm, rotated rx 180 ry 0 rz -180 deg; joints [-40.114, -26.652, 97.875, 69.09, 43.609, -62.181]
  MoveL 6315 to (-41.11, 53.34, 97.46) mm, rotated rx 180 ry 0 rz -180 deg; joints [-40.114, -26.652, 97.875, 69.09, 43.609, -62.181]
  Call Extruder(59.57665)
  MoveL 6316 to (-41.06, 52.75, 97.46) mm, rotated rx 180 ry 0 rz 180 deg; joints [-40.01, -26.698, 97.9, 68.999, 43.524, -62.101]
  MoveL 6317 to (-41.06, 52.75, 97.46) mm, rotated rx 180 ry 0 rz 180 deg; joints [-40.01, -26.698, 97.9, 68.999, 43.524, -62.101]
  Call Extruder(59.77292)
  MoveL 6318 to (-41.02, 52.37, 97.46) mm, rotated rx 180 ry 0 rz -180 deg; joints [-39.939, -26.727, 97.915, 68.938, 43.467, -62.048]
  MoveL 6319 to (-41.02, 52.37, 97.46) mm, rotated rx 180 ry 0 rz -180 deg; joints [-39.939, -26.727, 97.915, 68.938, 43.467, -62.048]
  Call Extruder(59.97006)
  MoveL 6320 to (-40.97, 51.98, 97.46) mm, rotated rx 180 ry 0 rz 180 deg; joints [-39.869, -26.756, 97.931, 68.876, 43.409, -61.995]
  MoveL 6321 to (-40.97, 51.98, 97.46) mm, rotated rx 180 ry 0 rz 180 deg; joints [-39.869, -26.756, 97.931, 68.876, 43.409, -61.995]
  Call Extruder(60.16807)
  MoveL 6322 to (-40.93, 51.59, 97.46) mm, rotated rx 180 ry 0 rz -180 deg; joints [-39.798, -26.784, 97.946, 68.815, 43.352, -61.942]
  MoveL 6323 to (-40.93, 51.59, 97.46) mm, rotated rx 180 ry 0 rz -180 deg; joints [-39.798, -26.784, 97.946, 68.815, 43.352, -61.942]
  Call Extruder(60.36695)
  MoveL 6324 to (-40.88, 51.2, 97.46) mm, rotated rx 180 ry 0 rz 180 deg; joints [-39.727, -26.813, 97.961, 68.753, 43.294, -61.889]
  MoveL 6325 to (-40.88, 51.2, 97.46) mm, rotated rx 180 ry 0 rz 180 deg; joints [-39.727, -26.813, 97.961, 68.753, 43.294, -61.889]
  Call Extruder(60.54602)
  MoveL 6326 to (-40.83, 50.86, 97.46) mm, rotated rx 180 ry 0 rz 180 deg; joints [-39.663, -26.838, 97.975, 68.697, 43.242, -61.841]
  MoveL 6327 to (-40.83, 50.86, 97.46) mm, rotated rx 180 ry 0 rz 180 deg; joints [-39.663, -26.838, 97.975, 68.697, 43.242, -61.841]
  Call Extruder(60.70520)
  MoveL 6328 to (-40.78, 50.55, 97.46) mm, rotated rx 180 ry 0 rz 180 deg; joints [-39.605, -26.859, 97.986, 68.648, 43.194, -61.798]
  MoveL 6329 to (-40.78, 50.55, 97.46) mm, rotated rx 180 ry 0 rz 180 deg; joints [-39.605, -26.859, 97.986, 68.648, 43.194, -61.798]
  Call Extruder(60.86511)
  MoveL 6330 to (-40.74, 50.24, 97.46) mm, rotated rx 180 ry 0 rz 180 deg; joints [-39.547, -26.88, 97.997, 68.598, 43.147, -61.756]
  MoveL 6331 to (-40.74, 50.24, 97.46) mm, rotated rx 180 ry 0 rz 180 deg; joints [-39.547, -26.88, 97.997, 68.598, 43.147, -61.756]
  Call Extruder(61.02575)
  MoveL 6332 to (-40.69, 49.94, 97.46) mm, rotated rx -180 ry 0 rz 180 deg; joints [-39.489, -26.901, 98.008, 68.548, 43.1, -61.713]
  MoveL 6333 to (-40.69, 49.94, 97.46) mm, rotated rx -180 ry 0 rz 180 deg; joints [-39.489, -26.901, 98.008, 68.548, 43.1, -61.713]
  Call Extruder(61.18711)
  MoveL 6334 to (-40.64, 49.63, 97.46) mm, rotated rx 180 ry 0 rz 180 deg; joints [-39.431, -26.922, 98.02, 68.498, 43.052, -61.67]
  MoveL 6335 to (-40.64, 49.63, 97.46) mm, rotated rx 180 ry 0 rz 180 deg; joints [-39.431, -26.922, 98.02, 68.498, 43.052, -61.67]
  Call Extruder(61.34921)
  MoveL 6336 to (-40.59, 49.33, 97.46) mm, rotated rx 180 ry 0 rz 180 deg; joints [-39.373, -26.943, 98.031, 68.448, 43.005, -61.627]
  MoveL 6337 to (-40.59, 49.33, 97.46) mm, rotated rx 180 ry 0 rz 180 deg; joints [-39.373, -26.943, 98.031, 68.448, 43.005, -61.627]
  Call Extruder(61.49740)
  MoveL 6338 to (-40.54, 49.05, 97.46) mm, rotated rx 180 ry 0 rz 180 deg; joints [-39.32, -26.962, 98.041, 68.402, 42.961, -61.588]
  MoveL 6339 to (-40.54, 49.05, 97.46) mm, rotated rx 180 ry 0 rz 180 deg; joints [-39.32, -26.962, 98.041, 68.402, 42.961, -61.588]
  Call Extruder(61.63163)
  MoveL 6340 to (-40.49, 48.8, 97.46) mm, rotated rx 180 ry 0 rz 180 deg; joints [-39.271, -26.978, 98.049, 68.36, 42.921, -61.553]
  MoveL 6341 to (-40.49, 48.8, 97.46) mm, rotated rx 180 ry 0 rz 180 deg; joints [-39.271, -26.978, 98.049, 68.36, 42.921, -61.553]
  Call Extruder(61.76647)
  MoveL 6342 to (-40.44, 48.55, 97.46) mm, rotated rx -180 ry 0 rz 180 deg; joints [-39.222, -26.994, 98.058, 68.319, 42.881, -61.518]
  MoveL 6343 to (-40.44, 48.55, 97.46) mm, rotated rx -180 ry 0 rz 180 deg; joints [-39.222, -26.994, 98.058, 68.319, 42.881, -61.518]
  Call Extruder(61.90192)
  MoveL 6344 to (-40.39, 48.3, 97.46) mm, rotated rx -180 ry 0 rz 180 deg; joints [-39.174, -27.01, 98.066, 68.277, 42.841, -61.482]
  MoveL 6345 to (-40.39, 48.3, 97.46) mm, rotated rx -180 ry 0 rz 180 deg; joints [-39.174, -27.01, 98.066, 68.277, 42.841, -61.482]
  Call Extruder(62.03798)
  MoveL 6346 to (-40.34, 48.05, 97.46) mm, rotated rx -180 ry 0 rz -180 deg; joints [-39.125, -27.026, 98.075, 68.235, 42.8, -61.447]
  MoveL 6347 to (-40.34, 48.05, 97.46) mm, rotated rx -180 ry 0 rz -180 deg; joints [-39.125, -27.026, 98.075, 68.235, 42.8, -61.447]
  Call Extruder(62.17465)
  MoveL 6348 to (-40.29, 47.8, 97.46) mm, rotated rx 180 ry 0 rz 180 deg; joints [-39.076, -27.042, 98.083, 68.193, 42.76, -61.411]
  MoveL 6349 to (-40.29, 47.8, 97.46) mm, rotated rx 180 ry 0 rz 180 deg; joints [-39.076, -27.042, 98.083, 68.193, 42.76, -61.411]
  Call Extruder(62.31193)
  MoveL 6350 to (-40.24, 47.55, 97.46) mm, rotated rx 180 ry 0 rz 180 deg; joints [-39.027, -27.058, 98.092, 68.151, 42.72, -61.376]
  MoveL 6351 to (-40.24, 47.55, 97.46) mm, rotated rx 180 ry 0 rz 180 deg; joints [-39.027, -27.058, 98.092, 68.151, 42.72, -61.376]
  Call Extruder(62.43761)
  MoveL 6352 to (-40.2, 47.33, 97.46) mm, rotated rx 180 ry 0 rz 180 deg; joints [-38.982, -27.072, 98.099, 68.113, 42.683, -61.343]
  MoveL 6353 to (-40.2, 47.33, 97.46) mm, rotated rx 180 ry 0 rz 180 deg; joints [-38.982, -27.072, 98.099, 68.113, 42.683, -61.343]
  Call Extruder(62.55156)
  MoveL 6354 to (-40.15, 47.12, 97.46) mm, rotated rx 180 ry 0 rz 180 deg; joints [-38.941, -27.084, 98.106, 68.078, 42.649, -61.314]
  MoveL 6355 to (-40.15, 47.12, 97.46) mm, rotated rx 180 ry 0 rz 180 deg; joints [-38.941, -27.084, 98.106, 68.078, 42.649, -61.314]
  Call Extruder(62.66597)
  MoveL 6356 to (-40.11, 46.92, 97.46) mm, rotated rx 180 ry 0 rz 180 deg; joints [-38.9, -27.097, 98.113, 68.043, 42.616, -61.285]
  MoveL 6357 to (-40.11, 46.92, 97.46) mm, rotated rx 180 ry 0 rz 180 deg; joints [-38.9, -27.097, 98.113, 68.043, 42.616, -61.285]
  Call Extruder(62.78083)
  MoveL 6358 to (-40.06, 46.72, 97.46) mm, rotated rx 180 ry 0 rz 180 deg; joints [-38.859, -27.109, 98.119, 68.008, 42.582, -61.255]
  MoveL 6359 to (-40.06, 46.72, 97.46) mm, rotated rx 180 ry 0 rz 180 deg; joints [-38.859, -27.109, 98.119, 68.008, 42.582, -61.255]
  Call Extruder(62.89614)
  MoveL 6360 to (-40.02, 46.51, 97.46) mm, rotated rx 180 ry 0 rz 180 deg; joints [-38.819, -27.122, 98.126, 67.973, 42.549, -61.226]
  MoveL 6361 to (-40.02, 46.51, 97.46) mm, rotated rx 180 ry 0 rz 180 deg; joints [-38.819, -27.122, 98.126, 67.973, 42.549, -61.226]
  Call Extruder(63.02552)
  MoveL 6362 to (-39.95, 46.29, 97.46) mm, rotated rx 180 ry 0 rz 180 deg; joints [-38.771, -27.134, 98.132, 67.934, 42.509, -61.193]
  MoveL 6363 to (-39.95, 46.29, 97.46) mm, rotated rx 180 ry 0 rz 180 deg; joints [-38.771, -27.134, 98.132, 67.934, 42.509, -61.193]
  Call Extruder(63.15547)
  MoveL 6364 to (-39.88, 46.06, 97.46) mm, rotated rx 180 ry 0 rz -180 deg; joints [-38.724, -27.145, 98.138, 67.894, 42.47, -61.161]
  MoveL 6365 to (-39.88, 46.06, 97.46) mm, rotated rx 180 ry 0 rz -180 deg; joints [-38.724, -27.145, 98.138, 67.894, 42.47, -61.161]
  Call Extruder(63.28598)
  MoveL 6366 to (-39.81, 45.84, 97.46) mm, rotated rx -180 ry 0 rz 180 deg; joints [-38.677, -27.157, 98.145, 67.855, 42.43, -61.128]
  MoveL 6367 to (-39.81, 45.84, 97.46) mm, rotated rx -180 ry 0 rz 180 deg; joints [-38.677, -27.157, 98.145, 67.855, 42.43, -61.128]
  Call Extruder(63.41705)
  MoveL 6368 to (-39.75, 45.62, 97.46) mm, rotated rx 180 ry 0 rz -180 deg; joints [-38.629, -27.169, 98.151, 67.815, 42.391, -61.096]
  MoveL 6369 to (-39.75, 45.62, 97.46) mm, rotated rx 180 ry 0 rz -180 deg; joints [-38.629, -27.169, 98.151, 67.815, 42.391, -61.096]
  Call Extruder(63.53870)
  MoveL 6370 to (-39.68, 45.41, 97.46) mm, rotated rx -180 ry 0 rz 180 deg; joints [-38.585, -27.179, 98.156, 67.779, 42.354, -61.066]
  MoveL 6371 to (-39.68, 45.41, 97.46) mm, rotated rx -180 ry 0 rz 180 deg; joints [-38.585, -27.179, 98.156, 67.779, 42.354, -61.066]
  Call Extruder(63.65082)
  MoveL 6372 to (-39.62, 45.22, 97.46) mm, rotated rx 180 ry 0 rz -180 deg; joints [-38.544, -27.188, 98.161, 67.745, 42.32, -61.038]
  MoveL 6373 to (-39.62, 45.22, 97.46) mm, rotated rx 180 ry 0 rz -180 deg; joints [-38.544, -27.188, 98.161, 67.745, 42.32, -61.038]
  Call Extruder(63.76339)
  MoveL 6374 to (-39.56, 45.03, 97.46) mm, rotated rx 180 ry 0 rz 180 deg; joints [-38.504, -27.198, 98.166, 67.711, 42.286, -61.01]
  MoveL 6375 to (-39.56, 45.03, 97.46) mm, rotated rx 180 ry 0 rz 180 deg; joints [-38.504, -27.198, 98.166, 67.711, 42.286, -61.01]
  Call Extruder(63.87640)
  MoveL 6376 to (-39.5, 44.85, 97.46) mm, rotated rx -180 ry 0 rz -180 deg; joints [-38.463, -27.207, 98.171, 67.678, 42.253, -60.983]
  MoveL 6377 to (-39.5, 44.85, 97.46) mm, rotated rx -180 ry 0 rz -180 deg; joints [-38.463, -27.207, 98.171, 67.678, 42.253, -60.983]
  Call Extruder(63.98986)
  MoveL 6378 to (-39.44, 44.66, 97.46) mm, rotated rx 180 ry 0 rz 180 deg; joints [-38.422, -27.216, 98.176, 67.644, 42.219, -60.955]
  MoveL 6379 to (-39.44, 44.66, 97.46) mm, rotated rx 180 ry 0 rz 180 deg; joints [-38.422, -27.216, 98.176, 67.644, 42.219, -60.955]
  Call Extruder(64.13750)
  MoveL 6380 to (-39.35, 44.42, 97.46) mm, rotated rx 180 ry 0 rz 180 deg; joints [-38.369, -27.227, 98.181, 67.6, 42.174, -60.919]
  MoveL 6381 to (-39.35, 44.42, 97.46) mm, rotated rx 180 ry 0 rz 180 deg; joints [-38.369, -27.227, 98.181, 67.6, 42.174, -60.919]
  Call Extruder(64.31984)
  MoveL 6382 to (-39.22, 44.13, 97.46) mm, rotated rx 180 ry 0 rz 180 deg; joints [-38.302, -27.238, 98.187, 67.546, 42.117, -60.876]
  MoveL 6383 to (-39.22, 44.13, 97.46) mm, rotated rx 180 ry 0 rz 180 deg; joints [-38.302, -27.238, 98.187, 67.546, 42.117, -60.876]
  Call Extruder(64.50294)
  MoveL 6384 to (-39.11, 43.83, 97.46) mm, rotated rx 180 ry 0 rz 180 deg; joints [-38.236, -27.25, 98.194, 67.492, 42.061, -60.832]
  MoveL 6385 to (-39.11, 43.83, 97.46) mm, rotated rx 180 ry 0 rz 180 deg; joints [-38.236, -27.25, 98.194, 67.492, 42.061, -60.832]
  Call Extruder(64.66062)
  MoveL 6386 to (-39, 43.58, 97.46) mm, rotated rx 180 ry 0 rz 180 deg; joints [-38.178, -27.259, 98.199, 67.446, 42.013, -60.795]
  MoveL 6387 to (-39, 43.58, 97.46) mm, rotated rx 180 ry 0 rz 180 deg; joints [-38.178, -27.259, 98.199, 67.446, 42.013, -60.795]
  Call Extruder(64.81891)
  MoveL 6388 to (-38.89, 43.34, 97.46) mm, rotated rx 180 ry 0 rz 180 deg; joints [-38.121, -27.269, 98.203, 67.399, 41.965, -60.758]
  MoveL 6389 to (-38.89, 43.34, 97.46) mm, rotated rx 180 ry 0 rz 180 deg; joints [-38.121, -27.269, 98.203, 67.399, 41.965, -60.758]
  Call Extruder(65.00093)
  MoveL 6390 to (-38.75, 43.06, 97.46) mm, rotated rx 180 ry 0 rz 180 deg; joints [-38.054, -27.277, 98.208, 67.346, 41.908, -60.716]
  MoveL 6391 to (-38.75, 43.06, 97.46) mm, rotated rx 180 ry 0 rz 180 deg; joints [-38.054, -27.277, 98.208, 67.346, 41.908, -60.716]
  Call Extruder(65.20748)
  MoveL 6392 to (-38.57, 42.75, 97.46) mm, rotated rx -180 ry 0 rz 180 deg; joints [-37.977, -27.283, 98.211, 67.287, 41.842, -60.67]
  MoveL 6393 to (-38.57, 42.75, 97.46) mm, rotated rx -180 ry 0 rz 180 deg; joints [-37.977, -27.283, 98.211, 67.287, 41.842, -60.67]
  Call Extruder(65.41481)
  MoveL 6394 to (-38.4, 42.45, 97.46) mm, rotated rx 180 ry 0 rz 180 deg; joints [-37.901, -27.29, 98.215, 67.228, 41.777, -60.624]
  MoveL 6395 to (-38.4, 42.45, 97.46) mm, rotated rx 180 ry 0 rz 180 deg; joints [-37.901, -27.29, 98.215, 67.228, 41.777, -60.624]
  Call Extruder(65.62293)
  MoveL 6396 to (-38.22, 42.15, 97.46) mm, rotated rx 180 ry 0 rz 180 deg; joints [-37.825, -27.296, 98.218, 67.168, 41.712, -60.578]
  MoveL 6397 to (-38.22, 42.15, 97.46) mm, rotated rx 180 ry 0 rz 180 deg; joints [-37.825, -27.296, 98.218, 67.168, 41.712, -60.578]
  Call Extruder(65.74064)
  MoveL 6398 to (-38.12, 41.97, 97.46) mm, rotated rx 180 ry 0 rz 180 deg; joints [-37.782, -27.3, 98.22, 67.135, 41.675, -60.552]
  MoveL 6399 to (-38.12, 41.97, 97.46) mm, rotated rx 180 ry 0 rz 180 deg; joints [-37.782, -27.3, 98.22, 67.135, 41.675, -60.552]
  Call Extruder(66.07349)
  MoveL 6400 to (-37.79, 41.52, 97.46) mm, rotated rx 180 ry 0 rz 180 deg; joints [-37.659, -27.302, 98.221, 67.043, 41.568, -60.483]
  MoveL 6401 to (-37.79, 41.52, 97.46) mm, rotated rx 180 ry 0 rz 180 deg; joints [-37.659, -27.302, 98.221, 67.043, 41.568, -60.483]
  Call Extruder(66.40752)
  MoveL 6402 to (-37.47, 41.07, 97.46) mm, rotated rx -180 ry 0 rz -180 deg; joints [-37.537, -27.304, 98.222, 66.951, 41.462, -60.413]
  MoveL 6403 to (-37.47, 41.07, 97.46) mm, rotated rx -180 ry 0 rz -180 deg; joints [-37.537, -27.304, 98.222, 66.951, 41.462, -60.413]
  Call Extruder(66.57511)
  MoveL 6404 to (-37.3, 40.85, 97.46) mm, rotated rx 180 ry 0 rz -180 deg; joints [-37.475, -27.305, 98.223, 66.905, 41.409, -60.378]
  Call Extruder(67.40442)
  MoveL 6405 to (-36.39, 39.81, 97.46) mm, rotated rx 180 ry 0 rz 180 deg; joints [-37.173, -27.292, 98.216, 66.684, 41.144, -60.216]
  Call Extruder(68.03549)
  MoveL 6406 to (-35.61, 39.11, 97.46) mm, rotated rx 180 ry 0 rz 180 deg; joints [-36.947, -27.264, 98.201, 66.526, 40.943, -60.105]
  MoveL 6407 to (-35.61, 39.11, 97.46) mm, rotated rx 180 ry 0 rz 180 deg; joints [-36.947, -27.264, 98.201, 66.526, 40.943, -60.105]
  Call Extruder(68.23306)
  MoveL 6408 to (-35.35, 38.9, 97.46) mm, rotated rx 180 ry 0 rz 180 deg; joints [-36.876, -27.255, 98.196, 66.477, 40.88, -60.071]
  Call Extruder(68.56708)
  MoveL 6409 to (-34.9, 38.57, 97.46) mm, rotated rx -180 ry 0 rz 180 deg; joints [-36.759, -27.233, 98.184, 66.399, 40.774, -60.018]
  MoveL 6410 to (-34.9, 38.57, 97.46) mm, rotated rx -180 ry 0 rz 180 deg; joints [-36.759, -27.233, 98.184, 66.399, 40.774, -60.018]
  Call Extruder(68.89991)
  MoveL 6411 to (-34.45, 38.24, 97.46) mm, rotated rx -180 ry 0 rz -180 deg; joints [-36.642, -27.21, 98.173, 66.321, 40.669, -59.965]
  MoveL 6412 to (-34.45, 38.24, 97.46) mm, rotated rx -180 ry 0 rz -180 deg; joints [-36.642, -27.21, 98.173, 66.321, 40.669, -59.965]
  Call Extruder(69.07916)
  MoveL 6413 to (-34.21, 38.07, 97.46) mm, rotated rx 180 ry 0 rz 180 deg; joints [-36.579, -27.198, 98.166, 66.279, 40.612, -59.936]
  MoveL 6414 to (-34.21, 38.07, 97.46) mm, rotated rx 180 ry 0 rz 180 deg; joints [-36.579, -27.198, 98.166, 66.279, 40.612, -59.936]
  Call Extruder(69.28727)
  MoveL 6415 to (-33.9, 37.89, 97.46) mm, rotated rx -180 ry 0 rz 180 deg; joints [-36.509, -27.179, 98.156, 66.234, 40.547, -59.907]
  MoveL 6416 to (-33.9, 37.89, 97.46) mm, rotated rx -180 ry 0 rz 180 deg; joints [-36.509, -27.179, 98.156, 66.234, 40.547, -59.907]
  Call Extruder(69.49460)
  MoveL 6417 to (-33.6, 37.71, 97.46) mm, rotated rx 180 ry 0 rz 180 deg; joints [-36.439, -27.16, 98.146, 66.189, 40.483, -59.879]
  MoveL 6418 to (-33.6, 37.71, 97.46) mm, rotated rx 180 ry 0 rz 180 deg; joints [-36.439, -27.16, 98.146, 66.189, 40.483, -59.879]
  Call Extruder(69.70115)
  MoveL 6419 to (-33.29, 37.54, 97.46) mm, rotated rx 180 ry 0 rz 180 deg; joints [-36.368, -27.142, 98.136, 66.144, 40.418, -59.85]
  MoveL 6420 to (-33.29, 37.54, 97.46) mm, rotated rx 180 ry 0 rz 180 deg; joints [-36.368, -27.142, 98.136, 66.144, 40.418, -59.85]
  Call Extruder(69.90692)
  MoveL 6421 to (-32.99, 37.36, 97.46) mm, rotated rx -180 ry 0 rz 180 deg; joints [-36.298, -27.123, 98.126, 66.099, 40.354, -59.821]
  MoveL 6422 to (-32.99, 37.36, 97.46) mm, rotated rx -180 ry 0 rz 180 deg; joints [-36.298, -27.123, 98.126, 66.099, 40.354, -59.821]
  Call Extruder(70.06522)
  MoveL 6423 to (-32.74, 37.26, 97.46) mm, rotated rx 180 ry 0 rz 180 deg; joints [-36.247, -27.104, 98.117, 66.069, 40.306, -59.803]
  MoveL 6424 to (-32.74, 37.26, 97.46) mm, rotated rx 180 ry 0 rz 180 deg; joints [-36.247, -27.104, 98.117, 66.069, 40.306, -59.803]
  Call Extruder(70.22292)
  MoveL 6425 to (-32.49, 37.15, 97.46) mm, rotated rx 180 ry 0 rz 180 deg; joints [-36.196, -27.086, 98.107, 66.038, 40.259, -59.785]
  MoveL 6426 to (-32.49, 37.15, 97.46) mm, rotated rx 180 ry 0 rz 180 deg; joints [-36.196, -27.086, 98.107, 66.038, 40.259, -59.785]
  Call Extruder(70.39301)
  MoveL 6427 to (-32.22, 37.04, 97.46) mm, rotated rx 180 ry 0 rz 180 deg; joints [-36.141, -27.065, 98.096, 66.006, 40.208, -59.766]
  MoveL 6428 to (-32.22, 37.04, 97.46) mm, rotated rx 180 ry 0 rz 180 deg; joints [-36.141, -27.065, 98.096, 66.006, 40.208, -59.766]
  Call Extruder(70.57534)
  MoveL 6429 to (-31.93, 36.91, 97.46) mm, rotated rx 180 ry 0 rz 180 deg; joints [-36.082, -27.043, 98.084, 65.971, 40.153, -59.745]
  MoveL 6430 to (-31.93, 36.91, 97.46) mm, rotated rx 180 ry 0 rz 180 deg; joints [-36.082, -27.043, 98.084, 65.971, 40.153, -59.745]
  Call Extruder(70.75692)
  MoveL 6431 to (-31.64, 36.79, 97.46) mm, rotated rx 180 ry 0 rz 180 deg; joints [-36.023, -27.021, 98.073, 65.937, 40.098, -59.725]
  MoveL 6432 to (-31.64, 36.79, 97.46) mm, rotated rx 180 ry 0 rz 180 deg; joints [-36.023, -27.021, 98.073, 65.937, 40.098, -59.725]
  Call Extruder(70.87038)
  MoveL 6433 to (-31.45, 36.73, 97.46) mm, rotated rx 180 ry 0 rz 180 deg; joints [-35.989, -27.006, 98.064, 65.917, 40.065, -59.714]
  MoveL 6434 to (-31.45, 36.73, 97.46) mm, rotated rx 180 ry 0 rz 180 deg; joints [-35.989, -27.006, 98.064, 65.917, 40.065, -59.714]
  Call Extruder(70.98339)
  MoveL 6435 to (-31.26, 36.67, 97.46) mm, rotated rx 180 ry 0 rz 180 deg; joints [-35.954, -26.99, 98.056, 65.898, 40.031, -59.704]
  MoveL 6436 to (-31.26, 36.67, 97.46) mm, rotated rx 180 ry 0 rz 180 deg; joints [-35.954, -26.99, 98.056, 65.898, 40.031, -59.704]
  Call Extruder(71.09596)
  MoveL 6437 to (-31.07, 36.61, 97.46) mm, rotated rx -180 ry 0 rz 180 deg; joints [-35.919, -26.974, 98.048, 65.878, 39.998, -59.693]
  MoveL 6438 to (-31.07, 36.61, 97.46) mm, rotated rx -180 ry 0 rz 180 deg; joints [-35.919, -26.974, 98.048, 65.878, 39.998, -59.693]
  Call Extruder(71.20808)
  MoveL 6439 to (-30.88, 36.55, 97.46) mm, rotated rx -180 ry 0 rz 180 deg; joints [-35.884, -26.959, 98.039, 65.859, 39.965, -59.683]
  MoveL 6440 to (-30.88, 36.55, 97.46) mm, rotated rx -180 ry 0 rz 180 deg; joints [-35.884, -26.959, 98.039, 65.859, 39.965, -59.683]
  Call Extruder(71.31976)
  MoveL 6441 to (-30.69, 36.49, 97.46) mm, rotated rx 180 ry 0 rz 180 deg; joints [-35.849, -26.943, 98.031, 65.84, 39.932, -59.672]
  MoveL 6442 to (-30.69, 36.49, 97.46) mm, rotated rx 180 ry 0 rz 180 deg; joints [-35.849, -26.943, 98.031, 65.84, 39.932, -59.672]
  Call Extruder(71.45084)
  MoveL 6443 to (-30.47, 36.42, 97.46) mm, rotated rx 180 ry 0 rz 180 deg; joints [-35.809, -26.924, 98.021, 65.818, 39.894, -59.66]
  MoveL 6444 to (-30.47, 36.42, 97.46) mm, rotated rx 180 ry 0 rz 180 deg; joints [-35.809, -26.924, 98.021, 65.818, 39.894, -59.66]
  Call Extruder(71.58135)
  MoveL 6445 to (-30.25, 36.35, 97.46) mm, rotated rx 180 ry 0 rz 180 deg; joints [-35.768, -26.905, 98.011, 65.796, 39.855, -59.649]
  MoveL 6446 to (-30.25, 36.35, 97.46) mm, rotated rx 180 ry 0 rz 180 deg; joints [-35.768, -26.905, 98.011, 65.796, 39.855, -59.649]
  Call Extruder(71.71129)
  MoveL 6447 to (-30.02, 36.28, 97.46) mm, rotated rx 180 ry 0 rz 180 deg; joints [-35.728, -26.886, 98, 65.773, 39.817, -59.637]
  MoveL 6448 to (-30.02, 36.28, 97.46) mm, rotated rx 180 ry 0 rz 180 deg; joints [-35.728, -26.886, 98, 65.773, 39.817, -59.637]
  Call Extruder(71.84067)
  MoveL 6449 to (-29.8, 36.22, 97.46) mm, rotated rx -180 ry 0 rz 180 deg; joints [-35.688, -26.867, 97.99, 65.751, 39.778, -59.625]
  MoveL 6450 to (-29.8, 36.22, 97.46) mm, rotated rx -180 ry 0 rz 180 deg; joints [-35.688, -26.867, 97.99, 65.751, 39.778, -59.625]
  Call Extruder(71.96263)
  MoveL 6451 to (-29.59, 36.16, 97.46) mm, rotated rx 180 ry 0 rz 180 deg; joints [-35.651, -26.848, 97.98, 65.732, 39.743, -59.615]
  MoveL 6452 to (-29.59, 36.16, 97.46) mm, rotated rx 180 ry 0 rz 180 deg; joints [-35.651, -26.848, 97.98, 65.732, 39.743, -59.615]
  Call Extruder(72.07748)
  MoveL 6453 to (-29.38, 36.12, 97.46) mm, rotated rx 180 ry 0 rz 180 deg; joints [-35.617, -26.829, 97.97, 65.715, 39.71, -59.607]
  MoveL 6454 to (-29.38, 36.12, 97.46) mm, rotated rx 180 ry 0 rz 180 deg; joints [-35.617, -26.829, 97.97, 65.715, 39.71, -59.607]
  Call Extruder(72.19188)
  MoveL 6455 to (-29.18, 36.07, 97.46) mm, rotated rx 180 ry 0 rz 180 deg; joints [-35.584, -26.81, 97.96, 65.698, 39.678, -59.599]
  MoveL 6456 to (-29.18, 36.07, 97.46) mm, rotated rx 180 ry 0 rz 180 deg; joints [-35.584, -26.81, 97.96, 65.698, 39.678, -59.599]
  Call Extruder(72.30582)
  MoveL 6457 to (-28.97, 36.03, 97.46) mm, rotated rx 180 ry 0 rz 180 deg; joints [-35.55, -26.791, 97.95, 65.681, 39.645, -59.591]
  MoveL 6458 to (-28.97, 36.03, 97.46) mm, rotated rx 180 ry 0 rz 180 deg; joints [-35.55, -26.791, 97.95, 65.681, 39.645, -59.591]
  Call Extruder(72.41931)
  MoveL 6459 to (-28.77, 35.98, 97.46) mm, rotated rx -180 ry 0 rz 180 deg; joints [-35.517, -26.772, 97.94, 65.664, 39.613, -59.583]
  MoveL 6460 to (-28.77, 35.98, 97.46) mm, rotated rx -180 ry 0 rz 180 deg; joints [-35.517, -26.772, 97.94, 65.664, 39.613, -59.583]
  Call Extruder(72.55660)
  MoveL 6461 to (-28.52, 35.93, 97.46) mm, rotated rx 180 ry 0 rz 180 deg; joints [-35.477, -26.749, 97.927, 65.644, 39.574, -59.574]
  MoveL 6462 to (-28.52, 35.93, 97.46) mm, rotated rx 180 ry 0 rz 180 deg; joints [-35.477, -26.749, 97.927, 65.644, 39.574, -59.574]
  Call Extruder(72.69327)
  MoveL 6463 to (-28.27, 35.88, 97.46) mm, rotated rx 180 ry 0 rz 180 deg; joints [-35.437, -26.725, 97.915, 65.624, 39.535, -59.565]
  MoveL 6464 to (-28.27, 35.88, 97.46) mm, rotated rx 180 ry 0 rz 180 deg; joints [-35.437, -26.725, 97.915, 65.624, 39.535, -59.565]
  Call Extruder(72.82933)
  MoveL 6465 to (-28.02, 35.83, 97.46) mm, rotated rx 180 ry 0 rz 180 deg; joints [-35.397, -26.702, 97.902, 65.604, 39.496, -59.556]
  MoveL 6466 to (-28.02, 35.83, 97.46) mm, rotated rx 180 ry 0 rz 180 deg; joints [-35.397, -26.702, 97.902, 65.604, 39.496, -59.556]
  Call Extruder(72.96478)
  MoveL 6467 to (-27.77, 35.78, 97.46) mm, rotated rx 180 ry 0 rz 180 deg; joints [-35.357, -26.679, 97.889, 65.585, 39.457, -59.547]
  MoveL 6468 to (-27.77, 35.78, 97.46) mm, rotated rx 180 ry 0 rz 180 deg; joints [-35.357, -26.679, 97.889, 65.585, 39.457, -59.547]
  Call Extruder(73.09962)
  MoveL 6469 to (-27.52, 35.73, 97.46) mm, rotated rx 180 ry 0 rz 180 deg; joints [-35.317, -26.655, 97.877, 65.565, 39.418, -59.538]
  MoveL 6470 to (-27.52, 35.73, 97.46) mm, rotated rx 180 ry 0 rz 180 deg; joints [-35.317, -26.655, 97.877, 65.565, 39.418, -59.538]
  Call Extruder(73.23385)
  MoveL 6471 to (-27.28, 35.68, 97.46) mm, rotated rx 180 ry 0 rz 180 deg; joints [-35.277, -26.632, 97.864, 65.545, 39.379, -59.529]
  MoveL 6472 to (-27.28, 35.68, 97.46) mm, rotated rx 180 ry 0 rz 180 deg; joints [-35.277, -26.632, 97.864, 65.545, 39.379, -59.529]
  Call Extruder(73.36747)
  MoveL 6473 to (-27.03, 35.63, 97.46) mm, rotated rx 180 ry 0 rz 180 deg; joints [-35.238, -26.608, 97.851, 65.526, 39.341, -59.521]
  MoveL 6474 to (-27.03, 35.63, 97.46) mm, rotated rx 180 ry 0 rz 180 deg; joints [-35.238, -26.608, 97.851, 65.526, 39.341, -59.521]
  Call Extruder(73.52957)
  MoveL 6475 to (-26.72, 35.59, 97.46) mm, rotated rx 180 ry 0 rz 180 deg; joints [-35.191, -26.578, 97.835, 65.504, 39.295, -59.511]
  MoveL 6476 to (-26.72, 35.59, 97.46) mm, rotated rx 180 ry 0 rz 180 deg; joints [-35.191, -26.578, 97.835, 65.504, 39.295, -59.511]
  Call Extruder(73.69094)
  MoveL 6477 to (-26.41, 35.54, 97.46) mm, rotated rx 180 ry 0 rz -180 deg; joints [-35.145, -26.548, 97.819, 65.482, 39.249, -59.502]
  MoveL 6478 to (-26.41, 35.54, 97.46) mm, rotated rx 180 ry 0 rz -180 deg; joints [-35.145, -26.548, 97.819, 65.482, 39.249, -59.502]
  Call Extruder(73.85158)
  MoveL 6479 to (-26.11, 35.49, 97.46) mm, rotated rx 180 ry 0 rz 180 deg; joints [-35.098, -26.518, 97.803, 65.46, 39.204, -59.493]
  MoveL 6480 to (-26.11, 35.49, 97.46) mm, rotated rx 180 ry 0 rz 180 deg; joints [-35.098, -26.518, 97.803, 65.46, 39.204, -59.493]
  Call Extruder(74.01150)
  MoveL 6481 to (-25.8, 35.44, 97.46) mm, rotated rx 180 ry 0 rz 180 deg; joints [-35.052, -26.488, 97.787, 65.438, 39.158, -59.484]
  MoveL 6482 to (-25.8, 35.44, 97.46) mm, rotated rx 180 ry 0 rz 180 deg; joints [-35.052, -26.488, 97.787, 65.438, 39.158, -59.484]
  Call Extruder(74.17068)
  MoveL 6483 to (-25.5, 35.39, 97.46) mm, rotated rx 180 ry 0 rz 180 deg; joints [-35.006, -26.458, 97.771, 65.416, 39.113, -59.475]
  MoveL 6484 to (-25.5, 35.39, 97.46) mm, rotated rx 180 ry 0 rz 180 deg; joints [-35.006, -26.458, 97.771, 65.416, 39.113, -59.475]
  Call Extruder(74.32914)
  MoveL 6485 to (-25.19, 35.34, 97.46) mm, rotated rx 180 ry 0 rz 180 deg; joints [-34.96, -26.428, 97.754, 65.395, 39.067, -59.466]
  MoveL 6486 to (-25.19, 35.34, 97.46) mm, rotated rx 180 ry 0 rz 180 deg; joints [-34.96, -26.428, 97.754, 65.395, 39.067, -59.466]
  Call Extruder(74.52802)
  MoveL 6487 to (-24.8, 35.3, 97.46) mm, rotated rx 180 ry 0 rz 180 deg; joints [-34.904, -26.389, 97.733, 65.37, 39.012, -59.458]
  MoveL 6488 to (-24.8, 35.3, 97.46) mm, rotated rx 180 ry 0 rz 180 deg; joints [-34.904, -26.389, 97.733, 65.37, 39.012, -59.458]
  Call Extruder(74.72603)
  MoveL 6489 to (-24.42, 35.25, 97.46) mm, rotated rx 180 ry 0 rz 180 deg; joints [-34.849, -26.35, 97.712, 65.345, 38.957, -59.449]
  MoveL 6490 to (-24.42, 35.25, 97.46) mm, rotated rx 180 ry 0 rz 180 deg; joints [-34.849, -26.35, 97.712, 65.345, 38.957, -59.449]
  Call Extruder(74.92317)
  MoveL 6491 to (-24.03, 35.21, 97.46) mm, rotated rx 180 ry 0 rz 180 deg; joints [-34.794, -26.311, 97.69, 65.321, 38.902, -59.44]
  MoveL 6492 to (-24.03, 35.21, 97.46) mm, rotated rx 180 ry 0 rz 180 deg; joints [-34.794, -26.311, 97.69, 65.321, 38.902, -59.44]
  Call Extruder(75.11944)
  MoveL 6493 to (-23.64, 35.16, 97.46) mm, rotated rx 180 ry 0 rz 180 deg; joints [-34.738, -26.271, 97.669, 65.296, 38.846, -59.431]
  MoveL 6494 to (-23.64, 35.16, 97.46) mm, rotated rx 180 ry 0 rz 180 deg; joints [-34.738, -26.271, 97.669, 65.296, 38.846, -59.431]
  Call Extruder(75.36513)
  MoveL 6495 to (-23.15, 35.11, 97.46) mm, rotated rx 180 ry 0 rz 180 deg; joints [-34.671, -26.221, 97.641, 65.267, 38.779, -59.422]
  MoveL 6496 to (-23.15, 35.11, 97.46) mm, rotated rx 180 ry 0 rz 180 deg; joints [-34.671, -26.221, 97.641, 65.267, 38.779, -59.422]
  Call Extruder(75.65986)
  MoveL 6497 to (-22.56, 35.07, 97.46) mm, rotated rx -180 ry 0 rz 180 deg; joints [-34.592, -26.159, 97.607, 65.235, 38.699, -59.412]
  MoveL 6498 to (-22.56, 35.07, 97.46) mm, rotated rx -180 ry 0 rz 180 deg; joints [-34.592, -26.159, 97.607, 65.235, 38.699, -59.412]
  Call Extruder(75.95325)
  MoveL 6499 to (-21.97, 35.02, 97.46) mm, rotated rx 180 ry 0 rz 180 deg; joints [-34.512, -26.097, 97.573, 65.202, 38.619, -59.402]
  MoveL 6500 to (-21.97, 35.02, 97.46) mm, rotated rx 180 ry 0 rz 180 deg; joints [-34.512, -26.097, 97.573, 65.202, 38.619, -59.402]
  Call Extruder(76.38658)
  MoveL 6501 to (-21.1, 34.98, 97.46) mm, rotated rx 180 ry 0 rz 180 deg; joints [-34.399, -26.003, 97.522, 65.158, 38.504, -59.392]
  MoveL 6502 to (-21.1, 34.98, 97.46) mm, rotated rx 180 ry 0 rz 180 deg; joints [-34.399, -26.003, 97.522, 65.158, 38.504, -59.392]
  Call Extruder(76.95874)
  MoveL 6503 to (-19.94, 34.93, 97.46) mm, rotated rx 180 ry 0 rz 180 deg; joints [-34.253, -25.876, 97.452, 65.103, 38.354, -59.381]
  MoveL 6504 to (-19.94, 34.93, 97.46) mm, rotated rx 180 ry 0 rz 180 deg; joints [-34.253, -25.876, 97.452, 65.103, 38.354, -59.381]
  Call Extruder(77.38658)
  MoveL 6505 to (-19.06, 34.91, 97.46) mm, rotated rx -180 ry 0 rz 180 deg; joints [-34.146, -25.78, 97.399, 65.064, 38.244, -59.375]
  Call Extruder(194.03526)
  MoveL 6506 to (219.06, 34.91, 97.46) mm, rotated rx 180 ry 0 rz 180 deg; joints [-18.248, 6.069, 70.925, 55.684, 22.28, -53.587]
  MoveL 6507 to (219.06, 34.91, 97.46) mm, rotated rx 180 ry 0 rz 180 deg; joints [-18.248, 6.069, 70.925, 55.684, 22.28, -53.587]
  Call Extruder(194.75084)
  MoveL 6508 to (220.52, 34.95, 97.46) mm, rotated rx 180 ry 0 rz 180 deg; joints [-18.199, 6.301, 70.668, 55.558, 22.254, -53.463]
  MoveL 6509 to (220.52, 34.95, 97.46) mm, rotated rx 180 ry 0 rz 180 deg; joints [-18.199, 6.301, 70.668, 55.558, 22.254, -53.463]
  Call Extruder(195.32557)
  MoveL 6510 to (221.68, 35, 97.46) mm, rotated rx 180 ry 0 rz 180 deg; joints [-18.162, 6.488, 70.461, 55.459, 22.235, -53.364]
  MoveL 6511 to (221.68, 35, 97.46) mm, rotated rx 180 ry 0 rz 180 deg; joints [-18.162, 6.488, 70.461, 55.459, 22.235, -53.364]
  Call Extruder(195.61897)
  MoveL 6512 to (222.27, 35.04, 97.46) mm, rotated rx -180 ry 0 rz 180 deg; joints [-18.146, 6.584, 70.354, 55.412, 22.229, -53.317]
  MoveL 6513 to (222.27, 35.04, 97.46) mm, rotated rx -180 ry 0 rz 180 deg; joints [-18.146, 6.584, 70.354, 55.412, 22.229, -53.317]
  Call Extruder(195.91369)
  MoveL 6514 to (222.86, 35.09, 97.46) mm, rotated rx 180 ry 0 rz 180 deg; joints [-18.13, 6.68, 70.248, 55.364, 22.222, -53.27]
  MoveL 6515 to (222.86, 35.09, 97.46) mm, rotated rx 180 ry 0 rz 180 deg; joints [-18.13, 6.68, 70.248, 55.364, 22.222, -53.27]
  Call Extruder(196.20975)
  MoveL 6516 to (223.45, 35.14, 97.46) mm, rotated rx -180 ry 0 rz 180 deg; joints [-18.113, 6.777, 70.14, 55.316, 22.215, -53.222]
  MoveL 6517 to (223.45, 35.14, 97.46) mm, rotated rx -180 ry 0 rz 180 deg; joints [-18.113, 6.777, 70.14, 55.316, 22.215, -53.222]
  Call Extruder(196.40603)
  MoveL 6518 to (223.84, 35.18, 97.46) mm, rotated rx 180 ry 0 rz -180 deg; joints [-18.104, 6.841, 70.069, 55.287, 22.212, -53.193]
  MoveL 6519 to (223.84, 35.18, 97.46) mm, rotated rx 180 ry 0 rz -180 deg; joints [-18.104, 6.841, 70.069, 55.287, 22.212, -53.193]
  Call Extruder(196.60317)
  MoveL 6520 to (224.22, 35.23, 97.46) mm, rotated rx 180 ry 0 rz 180 deg; joints [-18.095, 6.905, 69.997, 55.258, 22.209, -53.163]
  MoveL 6521 to (224.22, 35.23, 97.46) mm, rotated rx 180 ry 0 rz 180 deg; joints [-18.095, 6.905, 69.997, 55.258, 22.209, -53.163]
  Call Extruder(196.80118)
  MoveL 6522 to (224.61, 35.27, 97.46) mm, rotated rx -180 ry 0 rz 180 deg; joints [-18.087, 6.969, 69.925, 55.229, 22.206, -53.134]
  MoveL 6523 to (224.61, 35.27, 97.46) mm, rotated rx -180 ry 0 rz 180 deg; joints [-18.087, 6.969, 69.925, 55.229, 22.206, -53.134]
  Call Extruder(197.00005)
  MoveL 6524 to (225, 35.32, 97.46) mm, rotated rx 180 ry 0 rz 180 deg; joints [-18.078, 7.034, 69.853, 55.199, 22.203, -53.104]
  MoveL 6525 to (225, 35.32, 97.46) mm, rotated rx 180 ry 0 rz 180 deg; joints [-18.078, 7.034, 69.853, 55.199, 22.203, -53.104]
  Call Extruder(197.17913)
  MoveL 6526 to (225.34, 35.37, 97.46) mm, rotated rx 180 ry 0 rz 180 deg; joints [-18.07, 7.091, 69.788, 55.174, 22.202, -53.078]
  MoveL 6527 to (225.34, 35.37, 97.46) mm, rotated rx 180 ry 0 rz 180 deg; joints [-18.07, 7.091, 69.788, 55.174, 22.202, -53.078]
  Call Extruder(197.33832)
  MoveL 6528 to (225.65, 35.42, 97.46) mm, rotated rx -180 ry 0 rz 180 deg; joints [-18.065, 7.143, 69.731, 55.152, 22.201, -53.057]
  MoveL 6529 to (225.65, 35.42, 97.46) mm, rotated rx -180 ry 0 rz 180 deg; joints [-18.065, 7.143, 69.731, 55.152, 22.201, -53.057]
  Call Extruder(197.49823)
  MoveL 6530 to (225.96, 35.46, 97.46) mm, rotated rx -180 ry 0 rz 180 deg; joints [-18.059, 7.194, 69.673, 55.13, 22.2, -53.034]
  MoveL 6531 to (225.96, 35.46, 97.46) mm, rotated rx -180 ry 0 rz 180 deg; joints [-18.059, 7.194, 69.673, 55.13, 22.2, -53.034]
  Call Extruder(197.65887)
  MoveL 6532 to (226.26, 35.51, 97.46) mm, rotated rx 180 ry 0 rz 180 deg; joints [-18.054, 7.246, 69.615, 55.109, 22.199, -53.013]
  MoveL 6533 to (226.26, 35.51, 97.46) mm, rotated rx 180 ry 0 rz 180 deg; joints [-18.054, 7.246, 69.615, 55.109, 22.199, -53.013]
  Call Extruder(197.82023)
  MoveL 6534 to (226.57, 35.56, 97.46) mm, rotated rx -180 ry 0 rz 180 deg; joints [-18.048, 7.297, 69.557, 55.087, 22.198, -52.99]
  MoveL 6535 to (226.57, 35.56, 97.46) mm, rotated rx -180 ry 0 rz 180 deg; joints [-18.048, 7.297, 69.557, 55.087, 22.198, -52.99]
  Call Extruder(197.98233)
  MoveL 6536 to (226.87, 35.61, 97.46) mm, rotated rx 180 ry 0 rz -180 deg; joints [-18.042, 7.349, 69.499, 55.065, 22.197, -52.968]
  MoveL 6537 to (226.87, 35.61, 97.46) mm, rotated rx 180 ry 0 rz -180 deg; joints [-18.042, 7.349, 69.499, 55.065, 22.197, -52.968]
  Call Extruder(198.13052)
  MoveL 6538 to (227.15, 35.66, 97.46) mm, rotated rx -180 ry 0 rz 180 deg; joints [-18.038, 7.396, 69.446, 55.046, 22.197, -52.949]
  MoveL 6539 to (227.15, 35.66, 97.46) mm, rotated rx -180 ry 0 rz 180 deg; joints [-18.038, 7.396, 69.446, 55.046, 22.197, -52.949]
  Call Extruder(198.26476)
  MoveL 6540 to (227.4, 35.71, 97.46) mm, rotated rx 180 ry 0 rz 180 deg; joints [-18.034, 7.439, 69.398, 55.03, 22.197, -52.932]
  MoveL 6541 to (227.4, 35.71, 97.46) mm, rotated rx 180 ry 0 rz 180 deg; joints [-18.034, 7.439, 69.398, 55.03, 22.197, -52.932]
  Call Extruder(198.39960)
  MoveL 6542 to (227.65, 35.76, 97.46) mm, rotated rx -180 ry 0 rz 180 deg; joints [-18.031, 7.481, 69.35, 55.013, 22.198, -52.915]
  MoveL 6543 to (227.65, 35.76, 97.46) mm, rotated rx -180 ry 0 rz 180 deg; joints [-18.031, 7.481, 69.35, 55.013, 22.198, -52.915]
  Call Extruder(198.53505)
  MoveL 6544 to (227.9, 35.81, 97.46) mm, rotated rx -180 ry 0 rz 180 deg; joints [-18.027, 7.524, 69.302, 54.997, 22.198, -52.898]
  MoveL 6545 to (227.9, 35.81, 97.46) mm, rotated rx -180 ry 0 rz 180 deg; joints [-18.027, 7.524, 69.302, 54.997, 22.198, -52.898]
  Call Extruder(198.67111)
  MoveL 6546 to (228.15, 35.86, 97.46) mm, rotated rx -180 ry 0 rz -180 deg; joints [-18.024, 7.566, 69.254, 54.981, 22.198, -52.881]
  MoveL 6547 to (228.15, 35.86, 97.46) mm, rotated rx -180 ry 0 rz -180 deg; joints [-18.024, 7.566, 69.254, 54.981, 22.198, -52.881]
  Call Extruder(198.80779)
  MoveL 6548 to (228.4, 35.91, 97.46) mm, rotated rx 180 ry 0 rz -180 deg; joints [-18.02, 7.609, 69.206, 54.964, 22.199, -52.864]
  MoveL 6549 to (228.4, 35.91, 97.46) mm, rotated rx 180 ry 0 rz -180 deg; joints [-18.02, 7.609, 69.206, 54.964, 22.199, -52.864]
  Call Extruder(198.94507)
  MoveL 6550 to (228.64, 35.96, 97.46) mm, rotated rx -180 ry 0 rz -180 deg; joints [-18.017, 7.652, 69.158, 54.947, 22.199, -52.847]
  MoveL 6551 to (228.64, 35.96, 97.46) mm, rotated rx -180 ry 0 rz -180 deg; joints [-18.017, 7.652, 69.158, 54.947, 22.199, -52.847]
  Call Extruder(199.07074)
  MoveL 6552 to (228.87, 36, 97.46) mm, rotated rx -180 ry 0 rz 180 deg; joints [-18.014, 7.691, 69.114, 54.932, 22.2, -52.832]
  MoveL 6553 to (228.87, 36, 97.46) mm, rotated rx -180 ry 0 rz 180 deg; joints [-18.014, 7.691, 69.114, 54.932, 22.2, -52.832]
  Call Extruder(199.18469)
  MoveL 6554 to (229.08, 36.05, 97.46) mm, rotated rx 180 ry 0 rz 180 deg; joints [-18.012, 7.726, 69.074, 54.919, 22.201, -52.818]
  MoveL 6555 to (229.08, 36.05, 97.46) mm, rotated rx 180 ry 0 rz 180 deg; joints [-18.012, 7.726, 69.074, 54.919, 22.201, -52.818]
  Call Extruder(199.29908)
  MoveL 6556 to (229.28, 36.09, 97.46) mm, rotated rx -180 ry 0 rz 180 deg; joints [-18.009, 7.761, 69.034, 54.906, 22.201, -52.805]
  MoveL 6557 to (229.28, 36.09, 97.46) mm, rotated rx -180 ry 0 rz 180 deg; joints [-18.009, 7.761, 69.034, 54.906, 22.201, -52.805]
  Call Extruder(199.41393)
  MoveL 6558 to (229.48, 36.14, 97.46) mm, rotated rx 180 ry 0 rz 180 deg; joints [-18.007, 7.797, 68.994, 54.893, 22.202, -52.791]
  MoveL 6559 to (229.48, 36.14, 97.46) mm, rotated rx 180 ry 0 rz 180 deg; joints [-18.007, 7.797, 68.994, 54.893, 22.202, -52.791]
  Call Extruder(199.52924)
  MoveL 6560 to (229.69, 36.18, 97.46) mm, rotated rx 180 ry 0 rz 180 deg; joints [-18.005, 7.832, 68.954, 54.88, 22.203, -52.777]
  MoveL 6561 to (229.69, 36.18, 97.46) mm, rotated rx 180 ry 0 rz 180 deg; joints [-18.005, 7.832, 68.954, 54.88, 22.203, -52.777]
  Call Extruder(199.65360)
  MoveL 6562 to (229.9, 36.25, 97.46) mm, rotated rx 180 ry 0 rz -180 deg; joints [-18.004, 7.87, 68.911, 54.869, 22.205, -52.765]
  MoveL 6563 to (229.9, 36.25, 97.46) mm, rotated rx 180 ry 0 rz -180 deg; joints [-18.004, 7.87, 68.911, 54.869, 22.205, -52.765]
  Call Extruder(199.77848)
  MoveL 6564 to (230.12, 36.31, 97.46) mm, rotated rx 180 ry 0 rz -180 deg; joints [-18.003, 7.908, 68.867, 54.857, 22.208, -52.753]
  MoveL 6565 to (230.12, 36.31, 97.46) mm, rotated rx 180 ry 0 rz -180 deg; joints [-18.003, 7.908, 68.867, 54.857, 22.208, -52.753]
  Call Extruder(199.90388)
  MoveL 6566 to (230.33, 36.38, 97.46) mm, rotated rx 180 ry 0 rz 180 deg; joints [-18.003, 7.946, 68.824, 54.846, 22.21, -52.742]
  MoveL 6567 to (230.33, 36.38, 97.46) mm, rotated rx 180 ry 0 rz 180 deg; joints [-18.003, 7.946, 68.824, 54.846, 22.21, -52.742]
  Call Extruder(200.02979)
  MoveL 6568 to (230.55, 36.44, 97.46) mm, rotated rx -180 ry 0 rz 180 deg; joints [-18.002, 7.985, 68.781, 54.835, 22.213, -52.729]
  MoveL 6569 to (230.55, 36.44, 97.46) mm, rotated rx -180 ry 0 rz 180 deg; joints [-18.002, 7.985, 68.781, 54.835, 22.213, -52.729]
  Call Extruder(200.11575)
  MoveL 6570 to (230.7, 36.49, 97.46) mm, rotated rx 180 ry 0 rz -180 deg; joints [-18.002, 8.011, 68.751, 54.828, 22.215, -52.722]
  MoveL 6571 to (230.7, 36.49, 97.46) mm, rotated rx 180 ry 0 rz -180 deg; joints [-18.002, 8.011, 68.751, 54.828, 22.215, -52.722]
  Call Extruder(200.22765)
  MoveL 6572 to (230.88, 36.55, 97.46) mm, rotated rx 180 ry 0 rz 180 deg; joints [-18.002, 8.044, 68.713, 54.819, 22.217, -52.712]
  MoveL 6573 to (230.88, 36.55, 97.46) mm, rotated rx 180 ry 0 rz 180 deg; joints [-18.002, 8.044, 68.713, 54.819, 22.217, -52.712]
  Call Extruder(200.33999)
  MoveL 6574 to (231.07, 36.61, 97.46) mm, rotated rx 180 ry 0 rz -180 deg; joints [-18.002, 8.078, 68.675, 54.809, 22.22, -52.702]
  MoveL 6575 to (231.07, 36.61, 97.46) mm, rotated rx 180 ry 0 rz -180 deg; joints [-18.002, 8.078, 68.675, 54.809, 22.22, -52.702]
  Call Extruder(200.45278)
  MoveL 6576 to (231.26, 36.67, 97.46) mm, rotated rx -180 ry 0 rz 180 deg; joints [-18.002, 8.112, 68.636, 54.8, 22.223, -52.692]
  MoveL 6577 to (231.26, 36.67, 97.46) mm, rotated rx -180 ry 0 rz 180 deg; joints [-18.002, 8.112, 68.636, 54.8, 22.223, -52.692]
  Call Extruder(200.56601)
  MoveL 6578 to (231.45, 36.73, 97.46) mm, rotated rx 180 ry 0 rz 180 deg; joints [-18.002, 8.146, 68.598, 54.791, 22.225, -52.682]
  MoveL 6579 to (231.45, 36.73, 97.46) mm, rotated rx 180 ry 0 rz 180 deg; joints [-18.002, 8.146, 68.598, 54.791, 22.225, -52.682]
  Call Extruder(200.67969)
  MoveL 6580 to (231.64, 36.79, 97.46) mm, rotated rx 180 ry 0 rz 180 deg; joints [-18.002, 8.179, 68.559, 54.781, 22.228, -52.672]
  MoveL 6581 to (231.64, 36.79, 97.46) mm, rotated rx 180 ry 0 rz 180 deg; joints [-18.002, 8.179, 68.559, 54.781, 22.228, -52.672]
  Call Extruder(200.86165)
  MoveL 6582 to (231.93, 36.91, 97.46) mm, rotated rx 180 ry 0 rz 180 deg; joints [-18.005, 8.233, 68.498, 54.771, 22.235, -52.66]
  MoveL 6583 to (231.93, 36.91, 97.46) mm, rotated rx 180 ry 0 rz 180 deg; joints [-18.005, 8.233, 68.498, 54.771, 22.235, -52.66]
  Call Extruder(201.04437)
  MoveL 6584 to (232.22, 37.03, 97.46) mm, rotated rx -180 ry 0 rz 180 deg; joints [-18.008, 8.287, 68.437, 54.76, 22.241, -52.647]
  MoveL 6585 to (232.22, 37.03, 97.46) mm, rotated rx -180 ry 0 rz 180 deg; joints [-18.008, 8.287, 68.437, 54.76, 22.241, -52.647]
  Call Extruder(201.21479)
  MoveL 6586 to (232.49, 37.15, 97.46) mm, rotated rx -180 ry 0 rz -180 deg; joints [-18.011, 8.337, 68.38, 54.751, 22.248, -52.637]
  MoveL 6587 to (232.49, 37.15, 97.46) mm, rotated rx -180 ry 0 rz -180 deg; joints [-18.011, 8.337, 68.38, 54.751, 22.248, -52.637]
  Call Extruder(201.37278)
  MoveL 6588 to (232.74, 37.26, 97.46) mm, rotated rx -180 ry 0 rz 180 deg; joints [-18.013, 8.383, 68.327, 54.742, 22.254, -52.627]
  MoveL 6589 to (232.74, 37.26, 97.46) mm, rotated rx -180 ry 0 rz 180 deg; joints [-18.013, 8.383, 68.327, 54.742, 22.254, -52.627]
  Call Extruder(201.53139)
  MoveL 6590 to (232.99, 37.36, 97.46) mm, rotated rx -180 ry 0 rz 180 deg; joints [-18.016, 8.429, 68.274, 54.734, 22.26, -52.616]
  MoveL 6591 to (232.99, 37.36, 97.46) mm, rotated rx -180 ry 0 rz 180 deg; joints [-18.016, 8.429, 68.274, 54.734, 22.26, -52.616]
  Call Extruder(201.73755)
  MoveL 6592 to (233.29, 37.54, 97.46) mm, rotated rx 180 ry 0 rz 180 deg; joints [-18.024, 8.488, 68.207, 54.73, 22.271, -52.611]
  MoveL 6593 to (233.29, 37.54, 97.46) mm, rotated rx 180 ry 0 rz 180 deg; joints [-18.024, 8.488, 68.207, 54.73, 22.271, -52.611]
  Call Extruder(201.94450)
  MoveL 6594 to (233.6, 37.71, 97.46) mm, rotated rx 180 ry 0 rz 180 deg; joints [-18.033, 8.546, 68.14, 54.726, 22.283, -52.605]
  MoveL 6595 to (233.6, 37.71, 97.46) mm, rotated rx 180 ry 0 rz 180 deg; joints [-18.033, 8.546, 68.14, 54.726, 22.283, -52.605]
  Call Extruder(202.15222)
  MoveL 6596 to (233.9, 37.89, 97.46) mm, rotated rx -180 ry 0 rz 180 deg; joints [-18.041, 8.605, 68.073, 54.723, 22.294, -52.598]
  MoveL 6597 to (233.9, 37.89, 97.46) mm, rotated rx -180 ry 0 rz 180 deg; joints [-18.041, 8.605, 68.073, 54.723, 22.294, -52.598]
  Call Extruder(202.36072)
  MoveL 6598 to (234.21, 38.07, 97.46) mm, rotated rx 180 ry 0 rz 180 deg; joints [-18.049, 8.664, 68.005, 54.719, 22.306, -52.592]
  MoveL 6599 to (234.21, 38.07, 97.46) mm, rotated rx 180 ry 0 rz 180 deg; joints [-18.049, 8.664, 68.005, 54.719, 22.306, -52.592]
  Call Extruder(202.54027)
  MoveL 6600 to (234.45, 38.24, 97.46) mm, rotated rx 180 ry 0 rz 180 deg; joints [-18.06, 8.713, 67.949, 54.721, 22.318, -52.592]
  MoveL 6601 to (234.45, 38.24, 97.46) mm, rotated rx 180 ry 0 rz 180 deg; joints [-18.06, 8.713, 67.949, 54.721, 22.318, -52.592]
  Call Extruder(202.87368)
  MoveL 6602 to (234.9, 38.57, 97.46) mm, rotated rx 180 ry 0 rz 180 deg; joints [-18.079, 8.805, 67.844, 54.725, 22.342, -52.592]
  MoveL 6603 to (234.9, 38.57, 97.46) mm, rotated rx 180 ry 0 rz 180 deg; joints [-18.079, 8.805, 67.844, 54.725, 22.342, -52.592]
  Call Extruder(203.20828)
  MoveL 6604 to (235.35, 38.9, 97.46) mm, rotated rx 180 ry 0 rz 180 deg; joints [-18.099, 8.896, 67.739, 54.729, 22.365, -52.591]
  Call Extruder(204.03623)
  MoveL 6605 to (236.39, 39.81, 97.46) mm, rotated rx 180 ry 0 rz 180 deg; joints [-18.16, 9.114, 67.487, 54.761, 22.433, -52.61]
  Call Extruder(204.86417)
  MoveL 6606 to (237.3, 40.85, 97.46) mm, rotated rx -180 ry 0 rz 180 deg; joints [-18.24, 9.32, 67.249, 54.823, 22.515, -52.657]
  Call Extruder(205.03147)
  MoveL 6607 to (237.47, 41.07, 97.46) mm, rotated rx 180 ry 0 rz -180 deg; joints [-18.258, 9.359, 67.204, 54.84, 22.533, -52.671]
  MoveL 6608 to (237.47, 41.07, 97.46) mm, rotated rx 180 ry 0 rz -180 deg; joints [-18.258, 9.359, 67.204, 54.84, 22.533, -52.671]
  Call Extruder(205.36489)
  MoveL 6609 to (237.79, 41.52, 97.46) mm, rotated rx 180 ry 0 rz 180 deg; joints [-18.295, 9.437, 67.113, 54.874, 22.57, -52.698]
  MoveL 6610 to (237.79, 41.52, 97.46) mm, rotated rx 180 ry 0 rz 180 deg; joints [-18.295, 9.437, 67.113, 54.874, 22.57, -52.698]
  Call Extruder(205.69712)
  MoveL 6611 to (238.12, 41.98, 97.46) mm, rotated rx 180 ry 0 rz 180 deg; joints [-18.332, 9.516, 67.021, 54.907, 22.606, -52.725]
  MoveL 6612 to (238.12, 41.98, 97.46) mm, rotated rx 180 ry 0 rz 180 deg; joints [-18.332, 9.516, 67.021, 54.907, 22.606, -52.725]
  Call Extruder(205.81481)
  MoveL 6613 to (238.22, 42.15, 97.46) mm, rotated rx -180 ry 0 rz -180 deg; joints [-18.346, 9.542, 66.992, 54.922, 22.62, -52.737]
  MoveL 6614 to (238.22, 42.15, 97.46) mm, rotated rx -180 ry 0 rz -180 deg; joints [-18.346, 9.542, 66.992, 54.922, 22.62, -52.737]
  Call Extruder(206.02254)
  MoveL 6615 to (238.4, 42.45, 97.46) mm, rotated rx 180 ry 0 rz 180 deg; joints [-18.373, 9.587, 66.939, 54.948, 22.645, -52.76]
  MoveL 6616 to (238.4, 42.45, 97.46) mm, rotated rx 180 ry 0 rz 180 deg; joints [-18.373, 9.587, 66.939, 54.948, 22.645, -52.76]
  Call Extruder(206.22948)
  MoveL 6617 to (238.57, 42.75, 97.46) mm, rotated rx -180 ry 0 rz -180 deg; joints [-18.399, 9.633, 66.886, 54.975, 22.671, -52.782]
  MoveL 6618 to (238.57, 42.75, 97.46) mm, rotated rx -180 ry 0 rz -180 deg; joints [-18.399, 9.633, 66.886, 54.975, 22.671, -52.782]
  Call Extruder(206.43565)
  MoveL 6619 to (238.75, 43.06, 97.46) mm, rotated rx 180 ry 0 rz -180 deg; joints [-18.425, 9.678, 66.833, 55.002, 22.696, -52.804]
  MoveL 6620 to (238.75, 43.06, 97.46) mm, rotated rx 180 ry 0 rz -180 deg; joints [-18.425, 9.678, 66.833, 55.002, 22.696, -52.804]
  Call Extruder(206.61734)
  MoveL 6621 to (238.89, 43.34, 97.46) mm, rotated rx -180 ry 0 rz -180 deg; joints [-18.45, 9.717, 66.788, 55.027, 22.719, -52.826]
  MoveL 6622 to (238.89, 43.34, 97.46) mm, rotated rx -180 ry 0 rz -180 deg; joints [-18.45, 9.717, 66.788, 55.027, 22.719, -52.826]
  Call Extruder(206.77535)
  MoveL 6623 to (239, 43.58, 97.46) mm, rotated rx 180 ry 0 rz 180 deg; joints [-18.472, 9.748, 66.751, 55.053, 22.74, -52.848]
  MoveL 6624 to (239, 43.58, 97.46) mm, rotated rx 180 ry 0 rz 180 deg; joints [-18.472, 9.748, 66.751, 55.053, 22.74, -52.848]
  Call Extruder(206.93276)
  MoveL 6625 to (239.11, 43.83, 97.46) mm, rotated rx 180 ry 0 rz 180 deg; joints [-18.495, 9.78, 66.715, 55.078, 22.761, -52.869]
  MoveL 6626 to (239.11, 43.83, 97.46) mm, rotated rx 180 ry 0 rz 180 deg; joints [-18.495, 9.78, 66.715, 55.078, 22.761, -52.869]
  Call Extruder(207.11547)
  MoveL 6627 to (239.23, 44.13, 97.46) mm, rotated rx 180 ry 0 rz 180 deg; joints [-18.522, 9.816, 66.673, 55.108, 22.786, -52.895]
  MoveL 6628 to (239.23, 44.13, 97.46) mm, rotated rx 180 ry 0 rz 180 deg; joints [-18.522, 9.816, 66.673, 55.108, 22.786, -52.895]
  Call Extruder(207.29743)
  MoveL 6629 to (239.35, 44.42, 97.46) mm, rotated rx 180 ry 0 rz 180 deg; joints [-18.549, 9.852, 66.631, 55.138, 22.811, -52.921]
  MoveL 6630 to (239.35, 44.42, 97.46) mm, rotated rx 180 ry 0 rz 180 deg; joints [-18.549, 9.852, 66.631, 55.138, 22.811, -52.921]
  Call Extruder(207.44476)
  MoveL 6631 to (239.44, 44.66, 97.46) mm, rotated rx 180 ry 0 rz -180 deg; joints [-18.571, 9.88, 66.598, 55.164, 22.831, -52.943]
  MoveL 6632 to (239.44, 44.66, 97.46) mm, rotated rx 180 ry 0 rz -180 deg; joints [-18.571, 9.88, 66.598, 55.164, 22.831, -52.943]
  Call Extruder(207.55800)
  MoveL 6633 to (239.5, 44.85, 97.46) mm, rotated rx 180 ry 0 rz -180 deg; joints [-18.589, 9.901, 66.573, 55.185, 22.848, -52.961]
  MoveL 6634 to (239.5, 44.85, 97.46) mm, rotated rx 180 ry 0 rz -180 deg; joints [-18.589, 9.901, 66.573, 55.185, 22.848, -52.961]
  Call Extruder(207.67079)
  MoveL 6635 to (239.56, 45.03, 97.46) mm, rotated rx 180 ry 0 rz -180 deg; joints [-18.607, 9.921, 66.549, 55.205, 22.864, -52.979]
  MoveL 6636 to (239.56, 45.03, 97.46) mm, rotated rx 180 ry 0 rz -180 deg; joints [-18.607, 9.921, 66.549, 55.205, 22.864, -52.979]
  Call Extruder(207.78314)
  MoveL 6637 to (239.62, 45.22, 97.46) mm, rotated rx -180 ry 0 rz 180 deg; joints [-18.625, 9.942, 66.525, 55.226, 22.88, -52.997]
  MoveL 6638 to (239.62, 45.22, 97.46) mm, rotated rx -180 ry 0 rz 180 deg; joints [-18.625, 9.942, 66.525, 55.226, 22.88, -52.997]
  Call Extruder(207.89504)
  MoveL 6639 to (239.68, 45.41, 97.46) mm, rotated rx -180 ry 0 rz -180 deg; joints [-18.642, 9.962, 66.501, 55.247, 22.896, -53.015]
  MoveL 6640 to (239.68, 45.41, 97.46) mm, rotated rx -180 ry 0 rz -180 deg; joints [-18.642, 9.962, 66.501, 55.247, 22.896, -53.015]
  Call Extruder(208.01644)
  MoveL 6641 to (239.75, 45.62, 97.46) mm, rotated rx -180 ry 0 rz 180 deg; joints [-18.662, 9.985, 66.475, 55.27, 22.914, -53.035]
  MoveL 6642 to (239.75, 45.62, 97.46) mm, rotated rx -180 ry 0 rz 180 deg; joints [-18.662, 9.985, 66.475, 55.27, 22.914, -53.035]
  Call Extruder(208.14723)
  MoveL 6643 to (239.82, 45.84, 97.46) mm, rotated rx 180 ry 0 rz 180 deg; joints [-18.683, 10.008, 66.447, 55.295, 22.933, -53.057]
  MoveL 6644 to (239.82, 45.84, 97.46) mm, rotated rx 180 ry 0 rz 180 deg; joints [-18.683, 10.008, 66.447, 55.295, 22.933, -53.057]
  Call Extruder(208.27745)
  MoveL 6645 to (239.88, 46.06, 97.46) mm, rotated rx -180 ry 0 rz 180 deg; joints [-18.705, 10.032, 66.42, 55.32, 22.953, -53.079]
  MoveL 6646 to (239.88, 46.06, 97.46) mm, rotated rx -180 ry 0 rz 180 deg; joints [-18.705, 10.032, 66.42, 55.32, 22.953, -53.079]
  Call Extruder(208.40711)
  MoveL 6647 to (239.95, 46.29, 97.46) mm, rotated rx 180 ry 0 rz 180 deg; joints [-18.726, 10.056, 66.392, 55.345, 22.972, -53.1]
  MoveL 6648 to (239.95, 46.29, 97.46) mm, rotated rx 180 ry 0 rz 180 deg; joints [-18.726, 10.056, 66.392, 55.345, 22.972, -53.1]
  Call Extruder(208.53621)
  MoveL 6649 to (240.02, 46.51, 97.46) mm, rotated rx 180 ry 0 rz -180 deg; joints [-18.747, 10.079, 66.364, 55.37, 22.991, -53.122]
  MoveL 6650 to (240.02, 46.51, 97.46) mm, rotated rx 180 ry 0 rz -180 deg; joints [-18.747, 10.079, 66.364, 55.37, 22.991, -53.122]
  Call Extruder(208.65126)
  MoveL 6651 to (240.06, 46.72, 97.46) mm, rotated rx 180 ry 0 rz 180 deg; joints [-18.767, 10.098, 66.342, 55.395, 23.009, -53.144]
  MoveL 6652 to (240.06, 46.72, 97.46) mm, rotated rx 180 ry 0 rz 180 deg; joints [-18.767, 10.098, 66.342, 55.395, 23.009, -53.144]
  Call Extruder(208.76586)
  MoveL 6653 to (240.11, 46.92, 97.46) mm, rotated rx 180 ry 0 rz -180 deg; joints [-18.787, 10.117, 66.32, 55.419, 23.027, -53.165]
  MoveL 6654 to (240.11, 46.92, 97.46) mm, rotated rx 180 ry 0 rz -180 deg; joints [-18.787, 10.117, 66.32, 55.419, 23.027, -53.165]
  Call Extruder(208.88001)
  MoveL 6655 to (240.15, 47.12, 97.46) mm, rotated rx 180 ry 0 rz 180 deg; joints [-18.807, 10.136, 66.298, 55.443, 23.045, -53.186]
  MoveL 6656 to (240.15, 47.12, 97.46) mm, rotated rx 180 ry 0 rz 180 deg; joints [-18.807, 10.136, 66.298, 55.443, 23.045, -53.186]
  Call Extruder(208.99371)
  MoveL 6657 to (240.2, 47.33, 97.46) mm, rotated rx -180 ry 0 rz 180 deg; joints [-18.827, 10.155, 66.276, 55.468, 23.063, -53.208]
  MoveL 6658 to (240.2, 47.33, 97.46) mm, rotated rx -180 ry 0 rz 180 deg; joints [-18.827, 10.155, 66.276, 55.468, 23.063, -53.208]
  Call Extruder(209.11912)
  MoveL 6659 to (240.24, 47.56, 97.46) mm, rotated rx -180 ry 0 rz 180 deg; joints [-18.85, 10.176, 66.252, 55.495, 23.083, -53.232]
  MoveL 6660 to (240.24, 47.56, 97.46) mm, rotated rx -180 ry 0 rz 180 deg; joints [-18.85, 10.176, 66.252, 55.495, 23.083, -53.232]
  Call Extruder(209.25610)
  MoveL 6661 to (240.29, 47.8, 97.46) mm, rotated rx 180 ry 0 rz 180 deg; joints [-18.874, 10.198, 66.225, 55.525, 23.105, -53.258]
  MoveL 6662 to (240.29, 47.8, 97.46) mm, rotated rx 180 ry 0 rz 180 deg; joints [-18.874, 10.198, 66.225, 55.525, 23.105, -53.258]
  Call Extruder(209.39246)
  MoveL 6663 to (240.34, 48.05, 97.46) mm, rotated rx 180 ry 0 rz 180 deg; joints [-18.899, 10.22, 66.199, 55.555, 23.126, -53.284]
  MoveL 6664 to (240.34, 48.05, 97.46) mm, rotated rx 180 ry 0 rz 180 deg; joints [-18.899, 10.22, 66.199, 55.555, 23.126, -53.284]
  Call Extruder(209.52822)
  MoveL 6665 to (240.39, 48.3, 97.46) mm, rotated rx 180 ry 0 rz 180 deg; joints [-18.923, 10.243, 66.173, 55.585, 23.148, -53.31]
  MoveL 6666 to (240.39, 48.3, 97.46) mm, rotated rx 180 ry 0 rz 180 deg; joints [-18.923, 10.243, 66.173, 55.585, 23.148, -53.31]
  Call Extruder(209.66337)
  MoveL 6667 to (240.44, 48.55, 97.46) mm, rotated rx -180 ry 0 rz 180 deg; joints [-18.948, 10.265, 66.147, 55.615, 23.17, -53.337]
  MoveL 6668 to (240.44, 48.55, 97.46) mm, rotated rx -180 ry 0 rz 180 deg; joints [-18.948, 10.265, 66.147, 55.615, 23.17, -53.337]
  Call Extruder(209.79791)
  MoveL 6669 to (240.49, 48.8, 97.46) mm, rotated rx 180 ry 0 rz 180 deg; joints [-18.973, 10.287, 66.121, 55.644, 23.192, -53.363]
  MoveL 6670 to (240.49, 48.8, 97.46) mm, rotated rx 180 ry 0 rz 180 deg; joints [-18.973, 10.287, 66.121, 55.644, 23.192, -53.363]
  Call Extruder(209.93183)
  MoveL 6671 to (240.54, 49.05, 97.46) mm, rotated rx 180 ry 0 rz 180 deg; joints [-18.997, 10.31, 66.094, 55.674, 23.214, -53.388]
  MoveL 6672 to (240.54, 49.05, 97.46) mm, rotated rx 180 ry 0 rz 180 deg; joints [-18.997, 10.31, 66.094, 55.674, 23.214, -53.388]
  Call Extruder(210.07970)
  MoveL 6673 to (240.59, 49.33, 97.46) mm, rotated rx 180 ry 0 rz -180 deg; joints [-19.025, 10.333, 66.066, 55.707, 23.239, -53.418]
  MoveL 6674 to (240.59, 49.33, 97.46) mm, rotated rx 180 ry 0 rz -180 deg; joints [-19.025, 10.333, 66.066, 55.707, 23.239, -53.418]
  Call Extruder(210.24144)
  MoveL 6675 to (240.64, 49.63, 97.46) mm, rotated rx -180 ry 0 rz 180 deg; joints [-19.055, 10.359, 66.036, 55.745, 23.266, -53.451]
  MoveL 6676 to (240.64, 49.63, 97.46) mm, rotated rx -180 ry 0 rz 180 deg; joints [-19.055, 10.359, 66.036, 55.745, 23.266, -53.451]
  Call Extruder(210.40246)
  MoveL 6677 to (240.69, 49.94, 97.46) mm, rotated rx 180 ry 0 rz 180 deg; joints [-19.086, 10.385, 66.006, 55.782, 23.293, -53.484]
  MoveL 6678 to (240.69, 49.94, 97.46) mm, rotated rx 180 ry 0 rz 180 deg; joints [-19.086, 10.385, 66.006, 55.782, 23.293, -53.484]
  Call Extruder(210.56275)
  MoveL 6679 to (240.74, 50.24, 97.46) mm, rotated rx 180 ry 0 rz 180 deg; joints [-19.116, 10.41, 65.976, 55.819, 23.32, -53.516]
  MoveL 6680 to (240.74, 50.24, 97.46) mm, rotated rx 180 ry 0 rz 180 deg; joints [-19.116, 10.41, 65.976, 55.819, 23.32, -53.516]
  Call Extruder(210.72231)
  MoveL 6681 to (240.78, 50.55, 97.46) mm, rotated rx -180 ry 0 rz 180 deg; joints [-19.146, 10.436, 65.946, 55.856, 23.347, -53.549]
  MoveL 6682 to (240.78, 50.55, 97.46) mm, rotated rx -180 ry 0 rz 180 deg; joints [-19.146, 10.436, 65.946, 55.856, 23.347, -53.549]
  Call Extruder(210.88114)
  MoveL 6683 to (240.83, 50.86, 97.46) mm, rotated rx -180 ry 0 rz 180 deg; joints [-19.177, 10.462, 65.916, 55.893, 23.374, -53.581]
  MoveL 6684 to (240.83, 50.86, 97.46) mm, rotated rx -180 ry 0 rz 180 deg; joints [-19.177, 10.462, 65.916, 55.893, 23.374, -53.581]
  Call Extruder(211.05982)
  MoveL 6685 to (240.88, 51.2, 97.46) mm, rotated rx 180 ry 0 rz 180 deg; joints [-19.212, 10.489, 65.883, 55.935, 23.404, -53.618]
  MoveL 6686 to (240.88, 51.2, 97.46) mm, rotated rx 180 ry 0 rz 180 deg; joints [-19.212, 10.489, 65.883, 55.935, 23.404, -53.618]
  Call Extruder(211.25826)
  MoveL 6687 to (240.92, 51.59, 97.46) mm, rotated rx 180 ry 0 rz 180 deg; joints [-19.251, 10.519, 65.847, 55.983, 23.439, -53.661]
  MoveL 6688 to (240.92, 51.59, 97.46) mm, rotated rx 180 ry 0 rz 180 deg; joints [-19.251, 10.519, 65.847, 55.983, 23.439, -53.661]
  Call Extruder(211.45583)
  MoveL 6689 to (240.97, 51.98, 97.46) mm, rotated rx 180 ry 0 rz -180 deg; joints [-19.29, 10.549, 65.812, 56.031, 23.473, -53.703]
  MoveL 6690 to (240.97, 51.98, 97.46) mm, rotated rx 180 ry 0 rz -180 deg; joints [-19.29, 10.549, 65.812, 56.031, 23.473, -53.703]
  Call Extruder(211.65254)
  MoveL 6691 to (241.02, 52.36, 97.46) mm, rotated rx -180 ry 0 rz -180 deg; joints [-19.329, 10.58, 65.776, 56.079, 23.508, -53.745]
  MoveL 6692 to (241.02, 52.36, 97.46) mm, rotated rx -180 ry 0 rz -180 deg; joints [-19.329, 10.58, 65.776, 56.079, 23.508, -53.745]
  Call Extruder(211.84838)
  MoveL 6693 to (241.06, 52.75, 97.46) mm, rotated rx 180 ry 0 rz -180 deg; joints [-19.368, 10.61, 65.741, 56.126, 23.543, -53.786]
  MoveL 6694 to (241.06, 52.75, 97.46) mm, rotated rx 180 ry 0 rz -180 deg; joints [-19.368, 10.61, 65.741, 56.126, 23.543, -53.786]
  Call Extruder(212.14382)
  MoveL 6695 to (241.11, 53.34, 97.46) mm, rotated rx -180 ry 0 rz 180 deg; joints [-19.428, 10.652, 65.691, 56.201, 23.595, -53.852]
  MoveL 6696 to (241.11, 53.34, 97.46) mm, rotated rx -180 ry 0 rz 180 deg; joints [-19.428, 10.652, 65.691, 56.201, 23.595, -53.852]
  Call Extruder(212.43792)
  MoveL 6697 to (241.15, 53.93, 97.46) mm, rotated rx 180 ry 0 rz 180 deg; joints [-19.488, 10.694, 65.641, 56.275, 23.648, -53.917]
  MoveL 6698 to (241.15, 53.93, 97.46) mm, rotated rx 180 ry 0 rz 180 deg; joints [-19.488, 10.694, 65.641, 56.275, 23.648, -53.917]
  Call Extruder(212.73070)
  MoveL 6699 to (241.2, 54.52, 97.46) mm, rotated rx 180 ry 0 rz -180 deg; joints [-19.548, 10.737, 65.591, 56.348, 23.701, -53.982]
  MoveL 6700 to (241.2, 54.52, 97.46) mm, rotated rx 180 ry 0 rz -180 deg; joints [-19.548, 10.737, 65.591, 56.348, 23.701, -53.982]
  Call Extruder(213.30415)
  MoveL 6701 to (241.25, 55.68, 97.46) mm, rotated rx -180 ry 0 rz 180 deg; joints [-19.668, 10.813, 65.5, 56.496, 23.806, -54.113]
  MoveL 6702 to (241.25, 55.68, 97.46) mm, rotated rx -180 ry 0 rz 180 deg; joints [-19.668, 10.813, 65.5, 56.496, 23.806, -54.113]
  Call Extruder(214.01798)
  MoveL 6703 to (241.29, 57.14, 97.46) mm, rotated rx 180 ry 0 rz 180 deg; joints [-19.819, 10.906, 65.39, 56.681, 23.938, -54.276]
  Call Extruder(256.08287)
  MoveL 6704 to (241.29, 142.86, 97.46) mm, rotated rx 180 ry 0 rz 180 deg; joints [-28.232, 17.412, 57.314, 63.865, 31.797, -60.002]
  Call Extruder(256.51129)
  MoveL 6705 to (241.27, 143.73, 97.46) mm, rotated rx 180 ry 0 rz 180 deg; joints [-28.313, 17.49, 57.212, 63.907, 31.878, -60.027]
  MoveL 6706 to (241.27, 143.73, 97.46) mm, rotated rx 180 ry 0 rz 180 deg; joints [-28.313, 17.49, 57.212, 63.907, 31.878, -60.027]
  Call Extruder(257.08474)
  MoveL 6707 to (241.23, 144.9, 97.46) mm, rotated rx -180 ry 0 rz 180 deg; joints [-28.421, 17.592, 57.08, 63.966, 31.985, -60.062]
  MoveL 6708 to (241.23, 144.9, 97.46) mm, rotated rx -180 ry 0 rz 180 deg; joints [-28.421, 17.592, 57.08, 63.966, 31.985, -60.062]
  Call Extruder(257.51908)
  MoveL 6709 to (241.18, 145.77, 97.46) mm, rotated rx 180 ry 0 rz 180 deg; joints [-28.503, 17.666, 56.983, 64.011, 32.066, -60.09]
  MoveL 6710 to (241.18, 145.77, 97.46) mm, rotated rx 180 ry 0 rz 180 deg; joints [-28.503, 17.666, 56.983, 64.011, 32.066, -60.09]
  Call Extruder(257.81319)
  MoveL 6711 to (241.13, 146.36, 97.46) mm, rotated rx 180 ry 0 rz 180 deg; joints [-28.559, 17.714, 56.921, 64.043, 32.121, -60.11]
  MoveL 6712 to (241.13, 146.36, 97.46) mm, rotated rx 180 ry 0 rz 180 deg; joints [-28.559, 17.714, 56.921, 64.043, 32.121, -60.11]
  Call Extruder(258.10863)
  MoveL 6713 to (241.09, 146.95, 97.46) mm, rotated rx 180 ry 0 rz 180 deg; joints [-28.615, 17.762, 56.858, 64.074, 32.176, -60.129]
  MoveL 6714 to (241.09, 146.95, 97.46) mm, rotated rx 180 ry 0 rz 180 deg; joints [-28.615, 17.762, 56.858, 64.074, 32.176, -60.129]
  Call Extruder(258.35489)
  MoveL 6715 to (241.04, 147.44, 97.46) mm, rotated rx 180 ry 0 rz 180 deg; joints [-28.662, 17.8, 56.808, 64.101, 32.221, -60.147]
  MoveL 6716 to (241.04, 147.44, 97.46) mm, rotated rx 180 ry 0 rz 180 deg; joints [-28.662, 17.8, 56.808, 64.101, 32.221, -60.147]
  Call Extruder(258.55159)
  MoveL 6717 to (240.99, 147.83, 97.46) mm, rotated rx 180 ry 0 rz 180 deg; joints [-28.7, 17.829, 56.77, 64.123, 32.258, -60.161]
  MoveL 6718 to (240.99, 147.83, 97.46) mm, rotated rx 180 ry 0 rz 180 deg; joints [-28.7, 17.829, 56.77, 64.123, 32.258, -60.161]
  Call Extruder(258.74917)
  MoveL 6719 to (240.95, 148.22, 97.46) mm, rotated rx -180 ry 0 rz 180 deg; joints [-28.737, 17.858, 56.732, 64.146, 32.294, -60.176]
  MoveL 6720 to (240.95, 148.22, 97.46) mm, rotated rx -180 ry 0 rz 180 deg; joints [-28.737, 17.858, 56.732, 64.146, 32.294, -60.176]
  Call Extruder(258.94761)
  MoveL 6721 to (240.9, 148.6, 97.46) mm, rotated rx -180 ry 0 rz 180 deg; joints [-28.774, 17.888, 56.694, 64.168, 32.331, -60.19]
  MoveL 6722 to (240.9, 148.6, 97.46) mm, rotated rx -180 ry 0 rz 180 deg; joints [-28.774, 17.888, 56.694, 64.168, 32.331, -60.19]
  Call Extruder(259.14692)
  MoveL 6723 to (240.86, 148.99, 97.46) mm, rotated rx 180 ry 0 rz 180 deg; joints [-28.812, 17.917, 56.656, 64.19, 32.367, -60.205]
  MoveL 6724 to (240.86, 148.99, 97.46) mm, rotated rx 180 ry 0 rz 180 deg; joints [-28.812, 17.917, 56.656, 64.19, 32.367, -60.205]
  Call Extruder(259.30575)
  MoveL 6725 to (240.81, 149.3, 97.46) mm, rotated rx 180 ry 0 rz 180 deg; joints [-28.842, 17.938, 56.629, 64.209, 32.396, -60.218]
  MoveL 6726 to (240.81, 149.3, 97.46) mm, rotated rx 180 ry 0 rz 180 deg; joints [-28.842, 17.938, 56.629, 64.209, 32.396, -60.218]
  Call Extruder(259.46531)
  MoveL 6727 to (240.76, 149.6, 97.46) mm, rotated rx 180 ry 0 rz 180 deg; joints [-28.872, 17.959, 56.602, 64.228, 32.425, -60.23]
  MoveL 6728 to (240.76, 149.6, 97.46) mm, rotated rx 180 ry 0 rz 180 deg; joints [-28.872, 17.959, 56.602, 64.228, 32.425, -60.23]
  Call Extruder(259.62559)
  MoveL 6729 to (240.71, 149.91, 97.46) mm, rotated rx 180 ry 0 rz 180 deg; joints [-28.902, 17.979, 56.574, 64.246, 32.454, -60.243]
  MoveL 6730 to (240.71, 149.91, 97.46) mm, rotated rx 180 ry 0 rz 180 deg; joints [-28.902, 17.979, 56.574, 64.246, 32.454, -60.243]
  Call Extruder(259.78661)
  MoveL 6731 to (240.66, 150.21, 97.46) mm, rotated rx 180 ry 0 rz -180 deg; joints [-28.932, 18, 56.547, 64.265, 32.483, -60.256]
  MoveL 6732 to (240.66, 150.21, 97.46) mm, rotated rx 180 ry 0 rz -180 deg; joints [-28.932, 18, 56.547, 64.265, 32.483, -60.256]
  Call Extruder(259.94835)
  MoveL 6733 to (240.61, 150.52, 97.46) mm, rotated rx 180 ry 0 rz 180 deg; joints [-28.962, 18.022, 56.519, 64.284, 32.512, -60.268]
  MoveL 6734 to (240.61, 150.52, 97.46) mm, rotated rx 180 ry 0 rz 180 deg; joints [-28.962, 18.022, 56.519, 64.284, 32.512, -60.268]
  Call Extruder(260.11082)
  MoveL 6735 to (240.57, 150.83, 97.46) mm, rotated rx 180 ry 0 rz 180 deg; joints [-28.993, 18.043, 56.492, 64.302, 32.541, -60.281]
  MoveL 6736 to (240.57, 150.83, 97.46) mm, rotated rx 180 ry 0 rz 180 deg; joints [-28.993, 18.043, 56.492, 64.302, 32.541, -60.281]
  Call Extruder(260.24475)
  MoveL 6737 to (240.52, 151.08, 97.46) mm, rotated rx 180 ry 0 rz 180 deg; joints [-29.017, 18.058, 56.471, 64.318, 32.564, -60.292]
  MoveL 6738 to (240.52, 151.08, 97.46) mm, rotated rx 180 ry 0 rz 180 deg; joints [-29.017, 18.058, 56.471, 64.318, 32.564, -60.292]
  Call Extruder(260.37929)
  MoveL 6739 to (240.47, 151.32, 97.46) mm, rotated rx -180 ry 0 rz 180 deg; joints [-29.043, 18.074, 56.451, 64.335, 32.588, -60.304]
  MoveL 6740 to (240.47, 151.32, 97.46) mm, rotated rx -180 ry 0 rz 180 deg; joints [-29.043, 18.074, 56.451, 64.335, 32.588, -60.304]
  Call Extruder(260.51443)
  MoveL 6741 to (240.42, 151.57, 97.46) mm, rotated rx 180 ry 0 rz 180 deg; joints [-29.067, 18.089, 56.431, 64.351, 32.612, -60.315]
  MoveL 6742 to (240.42, 151.57, 97.46) mm, rotated rx 180 ry 0 rz 180 deg; joints [-29.067, 18.089, 56.431, 64.351, 32.612, -60.315]
  Call Extruder(260.65019)
  MoveL 6743 to (240.37, 151.82, 97.46) mm, rotated rx 180 ry 0 rz 180 deg; joints [-29.092, 18.105, 56.41, 64.367, 32.636, -60.326]
  MoveL 6744 to (240.37, 151.82, 97.46) mm, rotated rx 180 ry 0 rz 180 deg; joints [-29.092, 18.105, 56.41, 64.367, 32.636, -60.326]
  Call Extruder(260.78656)
  MoveL 6745 to (240.32, 152.07, 97.46) mm, rotated rx -180 ry 0 rz 180 deg; joints [-29.117, 18.12, 56.39, 64.383, 32.659, -60.337]
  MoveL 6746 to (240.32, 152.07, 97.46) mm, rotated rx -180 ry 0 rz 180 deg; joints [-29.117, 18.12, 56.39, 64.383, 32.659, -60.337]
  Call Extruder(260.92354)
  MoveL 6747 to (240.27, 152.32, 97.46) mm, rotated rx -180 ry 0 rz 180 deg; joints [-29.142, 18.136, 56.37, 64.399, 32.683, -60.348]
  MoveL 6748 to (240.27, 152.32, 97.46) mm, rotated rx -180 ry 0 rz 180 deg; joints [-29.142, 18.136, 56.37, 64.399, 32.683, -60.348]
  Call Extruder(261.06113)
  MoveL 6749 to (240.22, 152.57, 97.46) mm, rotated rx 180 ry 0 rz -180 deg; joints [-29.167, 18.151, 56.349, 64.415, 32.707, -60.36]
  MoveL 6750 to (240.22, 152.57, 97.46) mm, rotated rx 180 ry 0 rz -180 deg; joints [-29.167, 18.151, 56.349, 64.415, 32.707, -60.36]
  Call Extruder(261.17482)
  MoveL 6751 to (240.17, 152.77, 97.46) mm, rotated rx 180 ry 0 rz 180 deg; joints [-29.188, 18.164, 56.333, 64.429, 32.727, -60.369]
  MoveL 6752 to (240.17, 152.77, 97.46) mm, rotated rx 180 ry 0 rz 180 deg; joints [-29.188, 18.164, 56.333, 64.429, 32.727, -60.369]
  Call Extruder(261.28897)
  MoveL 6753 to (240.13, 152.98, 97.46) mm, rotated rx 180 ry 0 rz -180 deg; joints [-29.209, 18.176, 56.317, 64.443, 32.746, -60.379]
  MoveL 6754 to (240.13, 152.98, 97.46) mm, rotated rx 180 ry 0 rz -180 deg; joints [-29.209, 18.176, 56.317, 64.443, 32.746, -60.379]
  Call Extruder(261.40358)
  MoveL 6755 to (240.08, 153.18, 97.46) mm, rotated rx -180 ry 0 rz 180 deg; joints [-29.229, 18.188, 56.301, 64.456, 32.766, -60.388]
  MoveL 6756 to (240.08, 153.18, 97.46) mm, rotated rx -180 ry 0 rz 180 deg; joints [-29.229, 18.188, 56.301, 64.456, 32.766, -60.388]
  Call Extruder(261.51863)
  MoveL 6757 to (240.04, 153.39, 97.46) mm, rotated rx 180 ry 0 rz 180 deg; joints [-29.25, 18.2, 56.285, 64.47, 32.785, -60.398]
  MoveL 6758 to (240.04, 153.39, 97.46) mm, rotated rx 180 ry 0 rz 180 deg; joints [-29.25, 18.2, 56.285, 64.47, 32.785, -60.398]
  Call Extruder(261.64086)
  MoveL 6759 to (239.98, 153.6, 97.46) mm, rotated rx 180 ry 0 rz 180 deg; joints [-29.272, 18.211, 56.271, 64.485, 32.806, -60.409]
  MoveL 6760 to (239.98, 153.6, 97.46) mm, rotated rx 180 ry 0 rz 180 deg; joints [-29.272, 18.211, 56.271, 64.485, 32.806, -60.409]
  Call Extruder(261.77052)
  MoveL 6761 to (239.92, 153.82, 97.46) mm, rotated rx 180 ry 0 rz -180 deg; joints [-29.296, 18.221, 56.257, 64.502, 32.828, -60.422]
  MoveL 6762 to (239.92, 153.82, 97.46) mm, rotated rx 180 ry 0 rz -180 deg; joints [-29.296, 18.221, 56.257, 64.502, 32.828, -60.422]
  Call Extruder(261.90074)
  MoveL 6763 to (239.85, 154.05, 97.46) mm, rotated rx -180 ry 0 rz 180 deg; joints [-29.319, 18.231, 56.244, 64.519, 32.85, -60.435]
  MoveL 6764 to (239.85, 154.05, 97.46) mm, rotated rx -180 ry 0 rz 180 deg; joints [-29.319, 18.231, 56.244, 64.519, 32.85, -60.435]
  Call Extruder(262.03153)
  MoveL 6765 to (239.78, 154.27, 97.46) mm, rotated rx 180 ry 0 rz 180 deg; joints [-29.343, 18.242, 56.231, 64.536, 32.872, -60.447]
  MoveL 6766 to (239.78, 154.27, 97.46) mm, rotated rx 180 ry 0 rz 180 deg; joints [-29.343, 18.242, 56.231, 64.536, 32.872, -60.447]
  Call Extruder(262.16289)
  MoveL 6767 to (239.71, 154.5, 97.46) mm, rotated rx 180 ry 0 rz -180 deg; joints [-29.366, 18.252, 56.218, 64.553, 32.893, -60.46]
  MoveL 6768 to (239.71, 154.5, 97.46) mm, rotated rx 180 ry 0 rz -180 deg; joints [-29.366, 18.252, 56.218, 64.553, 32.893, -60.46]
  Call Extruder(262.27479)
  MoveL 6769 to (239.65, 154.68, 97.46) mm, rotated rx 180 ry 0 rz 180 deg; joints [-29.386, 18.26, 56.207, 64.568, 32.912, -60.471]
  MoveL 6770 to (239.65, 154.68, 97.46) mm, rotated rx 180 ry 0 rz 180 deg; joints [-29.386, 18.26, 56.207, 64.568, 32.912, -60.471]
  Call Extruder(262.38714)
  MoveL 6771 to (239.59, 154.87, 97.46) mm, rotated rx -180 ry 0 rz -180 deg; joints [-29.406, 18.268, 56.197, 64.582, 32.93, -60.482]
  MoveL 6772 to (239.59, 154.87, 97.46) mm, rotated rx -180 ry 0 rz -180 deg; joints [-29.406, 18.268, 56.197, 64.582, 32.93, -60.482]
  Call Extruder(262.49993)
  MoveL 6773 to (239.53, 155.06, 97.46) mm, rotated rx -180 ry 0 rz -180 deg; joints [-29.426, 18.275, 56.187, 64.597, 32.949, -60.494]
  MoveL 6774 to (239.53, 155.06, 97.46) mm, rotated rx -180 ry 0 rz -180 deg; joints [-29.426, 18.275, 56.187, 64.597, 32.949, -60.494]
  Call Extruder(262.61316)
  MoveL 6775 to (239.47, 155.25, 97.46) mm, rotated rx -180 ry 0 rz 180 deg; joints [-29.446, 18.283, 56.176, 64.612, 32.967, -60.505]
  MoveL 6776 to (239.47, 155.25, 97.46) mm, rotated rx -180 ry 0 rz 180 deg; joints [-29.446, 18.283, 56.176, 64.612, 32.967, -60.505]
  Call Extruder(262.72684)
  MoveL 6777 to (239.41, 155.44, 97.46) mm, rotated rx -180 ry 0 rz 180 deg; joints [-29.466, 18.291, 56.166, 64.626, 32.986, -60.516]
  MoveL 6778 to (239.41, 155.44, 97.46) mm, rotated rx -180 ry 0 rz 180 deg; joints [-29.466, 18.291, 56.166, 64.626, 32.986, -60.516]
  Call Extruder(262.90880)
  MoveL 6779 to (239.29, 155.73, 97.46) mm, rotated rx -180 ry 0 rz 180 deg; joints [-29.499, 18.299, 56.156, 64.652, 33.015, -60.536]
